C05460=1033.712,281.637,380.636,171.073,44.335,158.518
C05461=1033.719,281.885,380.604,171.077,44.336,158.519
C05462=1033.726,282.133,380.573,171.081,44.336,158.519
C05463=1033.732,282.381,380.541,171.084,44.336,158.520
C05464=1033.739,282.629,380.510,171.088,44.337,158.520
C05465=1033.746,282.877,380.479,171.092,44.337,158.521
C05466=1033.753,283.125,380.447,171.095,44.338,158.521
C05467=1033.759,283.373,380.416,171.100,44.338,158.522
C05468=1033.766,283.621,380.384,171.103,44.339,158.522
C05469=1033.773,283.869,380.353,171.107,44.340,158.522
C05470=1033.779,284.116,380.321,171.111,44.339,158.523
C05471=1033.786,284.364,380.290,171.115,44.340,158.523
C05472=1033.793,284.612,380.259,171.118,44.341,158.524
C05473=1033.800,284.860,380.226,171.123,44.341,158.524
C05474=1033.807,285.107,380.195,171.126,44.342,158.525
C05475=1033.814,285.356,380.163,171.130,44.342,158.525
C05476=1033.821,285.604,380.132,171.134,44.343,158.526
C05477=1033.827,285.852,380.100,171.138,44.343,158.526
C05478=1033.834,286.100,380.069,171.141,44.344,158.527
C05479=1033.841,286.347,380.037,171.146,44.344,158.527
C05480=1033.848,286.595,380.005,171.149,44.344,158.527
C05481=1033.855,286.843,379.974,171.154,44.345,158.528
C05482=1033.861,287.091,379.942,171.157,44.346,158.529
C05483=1033.869,287.339,379.910,171.161,44.346,158.529
C05484=1033.876,287.587,379.879,171.165,44.347,158.530
C05485=1033.882,287.835,379.846,171.169,44.348,158.530
C05486=1033.889,288.082,379.814,171.172,44.348,158.530
C05487=1033.895,288.330,379.783,171.177,44.349,158.531
C05488=1033.902,288.578,379.751,171.181,44.349,158.531
C05489=1033.910,288.826,379.719,171.185,44.350,158.532
C05490=1033.917,289.074,379.688,171.189,44.350,158.532
C05491=1033.923,289.321,379.655,171.192,44.351,158.533
C05492=1033.930,289.569,379.623,171.197,44.351,158.533
C05493=1033.937,289.817,379.591,171.200,44.352,158.534
C05494=1033.944,290.065,379.559,171.204,44.352,158.534
C05495=1033.950,290.313,379.527,171.208,44.353,158.535
C05496=1033.957,290.561,379.495,171.212,44.354,158.535
C05497=1033.964,290.808,379.463,171.216,44.354,158.536
C05498=1033.971,291.056,379.432,171.220,44.355,158.536
C05499=1033.981,291.421,379.384,171.226,44.356,158.537
C05500=1033.991,291.785,379.336,171.232,44.357,158.538
C05501=1034.001,292.150,379.289,171.238,44.358,158.539
C05502=1034.012,292.514,379.242,171.243,44.359,158.539
C05503=1034.018,292.762,379.209,171.248,44.359,158.540
C05504=1034.025,293.010,379.178,171.251,44.360,158.540
C05505=1034.032,293.258,379.145,171.256,44.361,158.541
C05506=1034.039,293.505,379.113,171.260,44.362,158.542
C05507=1034.045,293.753,379.081,171.263,44.362,158.542
C05508=1034.052,294.002,379.048,171.268,44.363,158.542
C05509=1034.059,294.249,379.016,171.271,44.364,158.543
C05510=1034.066,294.496,378.984,171.276,44.364,158.544
C05511=1034.072,294.744,378.952,171.279,44.365,158.544
C05512=1034.080,294.992,378.919,171.284,44.366,158.545
C05513=1034.086,295.240,378.887,171.288,44.366,158.545
C05514=1034.092,295.488,378.854,171.293,44.368,158.546
C05515=1034.099,295.736,378.821,171.296,44.368,158.546
C05516=1034.106,295.983,378.789,171.300,44.369,158.547
C05517=1034.113,296.231,378.756,171.304,44.370,158.547
C05518=1034.120,296.479,378.723,171.308,44.370,158.548
C05519=1034.127,296.726,378.691,171.313,44.371,158.549
C05520=1034.133,296.974,378.658,171.316,44.372,158.549
C05521=1034.140,297.222,378.625,171.321,44.373,158.550
C05522=1034.146,297.470,378.592,171.324,44.374,158.550
C05523=1034.153,297.717,378.560,171.329,44.375,158.551
C05524=1034.160,297.965,378.527,171.333,44.375,158.551
C05525=1034.167,298.212,378.493,171.338,44.376,158.552
C05526=1034.174,298.460,378.461,171.341,44.377,158.553
C05527=1034.180,298.708,378.428,171.345,44.378,158.553
C05528=1034.187,298.955,378.395,171.350,44.379,158.554
C05529=1034.194,299.204,378.362,171.353,44.380,158.554
C05530=1034.201,299.451,378.330,171.358,44.381,158.555
C05531=1034.208,299.699,378.297,171.361,44.381,158.555
C05532=1034.214,299.946,378.263,171.366,44.382,158.556
C05533=1034.220,300.194,378.231,171.371,44.383,158.557
C05534=1034.228,300.442,378.198,171.374,44.384,158.557
C05535=1034.234,300.690,378.165,171.379,44.385,158.558
C05536=1034.242,300.937,378.132,171.383,44.386,158.558
C05537=1034.248,301.185,378.099,171.387,44.387,158.559
C05538=1034.256,301.433,378.066,171.391,44.388,158.560
C05539=1034.262,301.680,378.033,171.396,44.388,158.560
C05540=1034.269,301.928,378.000,171.400,44.389,158.561
C05541=1034.275,302.176,377.967,171.404,44.390,158.561
C05542=1034.283,302.424,377.935,171.408,44.391,158.562
C05543=1034.290,302.671,377.901,171.413,44.392,158.563
C05544=1034.296,302.919,377.868,171.416,44.393,158.563
C05545=1034.303,303.166,377.835,171.421,44.394,158.564
C05546=1034.311,303.414,377.802,171.426,44.395,158.564
C05547=1034.318,303.662,377.769,171.429,44.396,158.565
C05548=1034.324,303.909,377.735,171.434,44.396,158.565
C05549=1034.331,304.157,377.702,171.438,44.397,158.566
C05550=1034.338,304.404,377.669,171.442,44.398,158.567
C05551=1034.345,304.652,377.636,171.447,44.399,158.567
C05552=1034.352,304.900,377.603,171.451,44.400,158.568
C05553=1034.359,305.148,377.570,171.456,44.401,158.569
C05554=1034.366,305.395,377.536,171.459,44.402,158.569
C05555=1034.378,305.776,377.485,171.466,44.404,158.570
C05556=1034.388,306.158,377.434,171.473,44.405,158.571
C05557=1034.399,306.539,377.383,171.480,44.407,158.572
C05558=1034.410,306.921,377.331,171.487,44.408,158.573
C05559=1034.417,307.169,377.298,171.490,44.409,158.574
C05560=1034.423,307.416,377.265,171.495,44.410,158.574
C05561=1034.431,307.663,377.231,171.500,44.411,158.575
C05562=1034.438,307.911,377.198,171.503,44.412,158.575
C05563=1034.445,308.159,377.164,171.508,44.413,158.576
C05564=1034.452,308.406,377.131,171.513,44.414,158.577
C05565=1034.459,308.654,377.098,171.517,44.415,158.577
C05566=1034.467,308.902,377.065,171.522,44.416,158.578
C05567=1034.474,309.149,377.031,171.526,44.417,158.579
C05568=1034.481,309.396,376.997,171.531,44.418,158.579
C05569=1034.488,309.645,376.964,171.535,44.419,158.580
C05570=1034.495,309.892,376.930,171.539,44.420,158.581
C05571=1034.503,310.140,376.897,171.544,44.421,158.581
C05572=1034.510,310.387,376.863,171.548,44.422,158.582
C05573=1034.517,310.635,376.829,171.553,44.423,158.583
C05574=1034.524,310.882,376.796,171.557,44.424,158.583
C05575=1034.531,311.130,376.762,171.562,44.425,158.584
C05576=1034.538,311.378,376.730,171.566,44.426,158.585
C05577=1034.546,311.625,376.696,171.571,44.427,158.585
C05578=1034.552,311.873,376.661,171.576,44.428,158.586
C05579=1034.559,312.120,376.627,171.580,44.430,158.587
C05580=1034.566,312.368,376.593,171.584,44.431,158.587
C05581=1034.573,312.615,376.559,171.589,44.432,158.588
C05582=1034.580,312.863,376.525,171.593,44.433,158.589
C05583=1034.586,313.111,376.491,171.598,44.435,158.589
C05584=1034.593,313.357,376.457,171.603,44.436,158.590
C05585=1034.600,313.605,376.422,171.606,44.437,158.591
C05586=1034.607,313.853,376.388,171.611,44.438,158.591
C05587=1034.614,314.101,376.355,171.616,44.439,158.592
C05588=1034.621,314.348,376.319,171.621,44.440,158.593
C05589=1034.628,314.596,376.286,171.625,44.442,158.594
C05590=1034.635,314.844,376.251,171.630,44.443,158.594
C05591=1034.641,315.090,376.217,171.635,44.444,158.595
C05592=1034.649,315.338,376.183,171.638,44.445,158.596
C05593=1034.655,315.586,376.149,171.643,44.447,158.597
C05594=1034.663,315.833,376.114,171.648,44.448,158.597
C05595=1034.669,316.081,376.080,171.653,44.449,158.598
C05596=1034.677,316.328,376.045,171.657,44.451,158.599
C05597=1034.684,316.576,376.011,171.662,44.452,158.599
C05598=1034.690,316.823,375.977,171.667,44.453,158.600
C05599=1034.698,317.071,375.942,171.671,44.454,158.601
C05600=1034.704,317.319,375.908,171.675,44.456,158.602
C05601=1034.712,317.566,375.874,171.680,44.457,158.602
C05602=1034.718,317.814,375.839,171.685,44.458,158.603
C05603=1034.726,318.061,375.805,171.690,44.460,158.604
C05604=1034.733,318.308,375.771,171.695,44.461,158.605
C05605=1034.740,318.556,375.736,171.699,44.463,158.605
C05606=1034.747,318.803,375.702,171.704,44.463,158.606
C05607=1034.754,319.051,375.667,171.709,44.465,158.607
C05608=1034.761,319.298,375.632,171.713,44.466,158.608
C05609=1034.768,319.546,375.598,171.718,44.468,158.608
C05610=1034.775,319.793,375.563,171.723,44.469,158.609
C05611=1034.787,320.179,375.509,171.730,44.471,158.610
C05612=1034.797,320.566,375.455,171.737,44.473,158.611
C05613=1034.809,320.952,375.401,171.745,44.475,158.613
C05614=1034.820,321.338,375.346,171.753,44.477,158.614
C05615=1034.827,321.585,375.312,171.757,44.479,158.615
C05616=1034.834,321.834,375.277,171.762,44.480,158.615
C05617=1034.842,322.081,375.243,171.767,44.481,158.616
C05618=1034.848,322.328,375.207,171.772,44.483,158.617
C05619=1034.856,322.575,375.173,171.777,44.485,158.618
C05620=1034.863,322.822,375.138,171.782,44.485,158.618
C05621=1034.871,323.070,375.103,171.787,44.487,158.619
C05622=1034.878,323.318,375.069,171.792,44.489,158.620
C05623=1034.885,323.566,375.034,171.795,44.490,158.621
C05624=1034.892,323.813,374.999,171.800,44.491,158.622
C05625=1034.900,324.061,374.964,171.805,44.493,158.622
C05626=1034.907,324.308,374.929,171.810,44.494,158.623
C05627=1034.914,324.555,374.894,171.815,44.496,158.624
C05628=1034.922,324.803,374.859,171.820,44.497,158.625
C05629=1034.929,325.050,374.824,171.825,44.499,158.626
C05630=1034.936,325.297,374.790,171.830,44.500,158.626
C05631=1034.944,325.545,374.754,171.835,44.501,158.627
C05632=1034.951,325.792,374.720,171.840,44.503,158.628
C05633=1034.958,326.040,374.684,171.845,44.504,158.629
C05634=1034.966,326.287,374.650,171.850,44.506,158.630
C05635=1034.973,326.535,374.614,171.855,44.507,158.630
C05636=1034.981,326.783,374.579,171.860,44.509,158.631
C05637=1034.988,327.030,374.544,171.865,44.510,158.632
C05638=1034.996,327.276,374.509,171.870,44.512,158.633
C05639=1035.003,327.524,374.474,171.875,44.513,158.634
C05640=1035.010,327.772,374.439,171.880,44.515,158.635
C05641=1035.018,328.020,374.404,171.885,44.516,158.635
C05642=1035.025,328.267,374.369,171.890,44.517,158.636
C05643=1035.033,328.514,374.333,171.895,44.519,158.637
C05644=1035.040,328.761,374.298,171.900,44.521,158.638
C05645=1035.047,329.008,374.262,171.905,44.523,158.639
C05646=1035.054,329.256,374.226,171.910,44.524,158.640
C05647=1035.061,329.504,374.191,171.915,44.526,158.640
C05648=1035.069,329.751,374.155,171.920,44.528,158.641
C05649=1035.075,329.998,374.120,171.925,44.529,158.642
C05650=1035.083,330.246,374.084,171.930,44.531,158.643
C05651=1035.090,330.493,374.048,171.935,44.532,158.644
C05652=1035.097,330.741,374.012,171.941,44.534,158.645
C05653=1035.105,330.988,373.978,171.946,44.536,158.646
C05654=1035.113,331.235,373.941,171.951,44.538,158.646
C05655=1035.120,331.482,373.906,171.956,44.539,158.647
C05656=1035.127,331.730,373.870,171.961,44.541,158.648
C05657=1035.134,331.977,373.834,171.966,44.543,158.649
C05658=1035.142,332.225,373.799,171.971,44.544,158.650
C05659=1035.149,332.472,373.763,171.976,44.546,158.651
C05660=1035.156,332.719,373.727,171.981,44.548,158.652
C05661=1035.164,332.967,373.691,171.986,44.550,158.653
C05662=1035.171,333.214,373.655,171.991,44.551,158.654
C05663=1035.178,333.461,373.619,171.996,44.553,158.654
C05664=1035.185,333.708,373.583,172.002,44.555,158.655
C05665=1035.193,333.956,373.548,172.007,44.557,158.656
C05666=1035.201,334.204,373.512,172.012,44.558,158.657
C05667=1035.212,334.585,373.456,172.021,44.561,158.659
C05668=1035.223,334.966,373.401,172.028,44.564,158.660
C05669=1035.235,335.348,373.345,172.036,44.567,158.661
C05670=1035.246,335.729,373.289,172.045,44.570,158.663
C05671=1035.254,335.977,373.252,172.050,44.571,158.664
C05672=1035.261,336.224,373.216,172.055,44.573,158.665
C05673=1035.268,336.471,373.180,172.061,44.575,158.666
C05674=1035.275,336.719,373.143,172.066,44.577,158.667
C05675=1035.283,336.966,373.107,172.071,44.579,158.668
C05676=1035.290,337.213,373.071,172.076,44.581,158.668
C05677=1035.298,337.460,373.035,172.082,44.583,158.670
C05678=1035.305,337.708,372.999,172.088,44.585,158.671
C05679=1035.312,337.956,372.962,172.093,44.586,158.671
C05680=1035.319,338.202,372.926,172.098,44.588,158.672
C05681=1035.327,338.449,372.889,172.103,44.591,158.673
C05682=1035.335,338.697,372.853,172.108,44.592,158.674
C05683=1035.343,338.944,372.817,172.114,44.594,158.675
C05684=1035.350,339.192,372.780,172.120,44.596,158.676
C05685=1035.357,339.438,372.744,172.125,44.598,158.677
C05686=1035.365,339.685,372.707,172.130,44.600,158.678
C05687=1035.372,339.933,372.671,172.135,44.602,158.679
C05688=1035.379,340.181,372.634,172.142,44.604,158.680
C05689=1035.387,340.427,372.597,172.147,44.606,158.681
C05690=1035.395,340.675,372.561,172.152,44.608,158.682
C05691=1035.403,340.922,372.524,172.157,44.610,158.683
C05692=1035.410,341.170,372.487,172.164,44.612,158.684
C05693=1035.417,341.416,372.452,172.169,44.614,158.685
C05694=1035.425,341.663,372.415,172.174,44.616,158.686
C05695=1035.432,341.910,372.377,172.179,44.618,158.687
C05696=1035.440,342.158,372.341,172.185,44.620,158.688
C05697=1035.447,342.405,372.303,172.191,44.622,158.689
C05698=1035.455,342.652,372.267,172.196,44.624,158.690
C05699=1035.462,342.899,372.230,172.201,44.626,158.691
C05700=1035.470,343.146,372.193,172.207,44.628,158.692
C05701=1035.477,343.394,372.156,172.213,44.631,158.693
C05702=1035.485,343.641,372.119,172.219,44.633,158.694
C05703=1035.492,343.888,372.081,172.224,44.635,158.696
C05704=1035.500,344.135,372.045,172.230,44.637,158.697
C05705=1035.507,344.382,372.008,172.235,44.639,158.698
C05706=1035.515,344.629,371.971,172.241,44.641,158.699
C05707=1035.522,344.876,371.933,172.246,44.643,158.700
C05708=1035.530,345.124,371.897,172.252,44.645,158.701
C05709=1035.537,345.371,371.859,172.258,44.647,158.702
C05710=1035.545,345.618,371.823,172.263,44.650,158.703
C05711=1035.552,345.865,371.785,172.269,44.652,158.704
C05712=1035.560,346.112,371.748,172.275,44.654,158.705
C05713=1035.568,346.359,371.711,172.280,44.656,158.706
C05714=1035.575,346.606,371.673,172.287,44.659,158.707
C05715=1035.583,346.854,371.636,172.292,44.661,158.708
C05716=1035.591,347.101,371.598,172.297,44.663,158.709
C05717=1035.599,347.348,371.561,172.303,44.665,158.710
C05718=1035.606,347.595,371.524,172.309,44.668,158.712
C05719=1035.614,347.842,371.487,172.315,44.670,158.713
C05720=1035.621,348.089,371.449,172.321,44.672,158.714
C05721=1035.629,348.337,371.411,172.326,44.675,158.715
C05722=1035.637,348.583,371.374,172.332,44.676,158.716
C05723=1035.649,348.961,371.317,172.342,44.680,158.717
C05724=1035.660,349.339,371.259,172.350,44.684,158.719
C05725=1035.672,349.718,371.202,172.359,44.687,158.721
C05726=1035.684,350.096,371.144,172.368,44.691,158.723
C05727=1035.691,350.343,371.107,172.374,44.693,158.724
C05728=1035.699,350.590,371.068,172.380,44.696,158.725
C05729=1035.706,350.837,371.030,172.385,44.698,158.726
C05730=1035.715,351.084,370.993,172.391,44.700,158.727
C05731=1035.722,351.331,370.955,172.398,44.703,158.728
C05732=1035.730,351.579,370.917,172.403,44.705,158.729
C05733=1035.737,351.825,370.879,172.409,44.708,158.731
C05734=1035.745,352.072,370.842,172.415,44.710,158.732
C05735=1035.753,352.319,370.803,172.422,44.713,158.733
C05736=1035.761,352.566,370.766,172.427,44.715,158.734
C05737=1035.769,352.813,370.728,172.433,44.717,158.735
C05738=1035.776,353.060,370.689,172.439,44.720,158.737
C05739=1035.784,353.307,370.652,172.446,44.723,158.738
C05740=1035.792,353.554,370.613,172.451,44.725,158.739
C05741=1035.799,353.801,370.575,172.457,44.727,158.740
C05742=1035.807,354.049,370.537,172.463,44.730,158.741
C05743=1035.815,354.295,370.499,172.470,44.732,158.743
C05744=1035.823,354.541,370.461,172.475,44.735,158.744
C05745=1035.831,354.789,370.423,172.482,44.738,158.745
C05746=1035.838,355.036,370.385,172.488,44.740,158.746
C05747=1035.847,355.283,370.346,172.494,44.742,158.747
C05748=1035.854,355.529,370.308,172.500,44.745,158.748
C05749=1035.862,355.777,370.270,172.506,44.747,158.750
C05750=1035.869,356.024,370.232,172.512,44.750,158.751
C05751=1035.878,356.271,370.193,172.518,44.752,158.752
C05752=1035.885,356.518,370.155,172.524,44.755,158.753
C05753=1035.893,356.765,370.117,172.531,44.758,158.755
C05754=1035.901,357.012,370.078,172.537,44.761,158.756
C05755=1035.909,357.258,370.040,172.543,44.763,158.757
C05756=1035.917,357.506,370.001,172.549,44.766,158.758
C05757=1035.925,357.752,369.963,172.555,44.768,158.760
C05758=1035.933,357.999,369.923,172.562,44.771,158.761
C05759=1035.941,358.245,369.885,172.568,44.774,158.762
C05760=1035.949,358.493,369.847,172.574,44.777,158.763
C05761=1035.957,358.740,369.808,172.581,44.779,158.765
C05762=1035.965,358.986,369.770,172.587,44.782,158.766
C05763=1035.973,359.233,369.731,172.593,44.784,158.767
C05764=1035.981,359.480,369.692,172.600,44.787,158.769
C05765=1035.988,359.727,369.653,172.606,44.790,158.770
C05766=1035.996,359.974,369.614,172.612,44.792,158.771
C05767=1036.005,360.221,369.575,172.619,44.795,158.772
C05768=1036.012,360.467,369.537,172.625,44.798,158.774
C05769=1036.020,360.714,369.498,172.631,44.801,158.775
C05770=1036.029,360.961,369.459,172.638,44.804,158.776
C05771=1036.037,361.208,369.420,172.644,44.807,158.778
C05772=1036.044,361.455,369.382,172.650,44.809,158.779
C05773=1036.052,361.702,369.342,172.657,44.812,158.780
C05774=1036.061,361.948,369.303,172.664,44.815,158.782
C05775=1036.069,362.196,369.264,172.670,44.818,158.783
C05776=1036.076,362.442,369.225,172.676,44.821,158.784
C05777=1036.084,362.689,369.186,172.683,44.824,158.786
C05778=1036.092,362.936,369.146,172.690,44.827,158.787
C05779=1036.104,363.320,369.086,172.699,44.831,158.789
C05780=1036.117,363.704,369.024,172.709,44.836,158.791
C05781=1036.129,364.089,368.963,172.720,44.840,158.793
C05782=1036.142,364.473,368.901,172.730,44.845,158.795
C05783=1036.150,364.720,368.862,172.736,44.848,158.797
C05784=1036.158,364.967,368.822,172.743,44.851,158.798
C05785=1036.166,365.214,368.783,172.750,44.854,158.800
C05786=1036.174,365.461,368.743,172.757,44.857,158.801
C05787=1036.182,365.707,368.704,172.763,44.860,158.802
C05788=1036.191,365.954,368.665,172.770,44.863,158.804
C05789=1036.199,366.201,368.625,172.777,44.866,158.805
C05790=1036.207,366.447,368.586,172.783,44.869,158.807
C05791=1036.215,366.694,368.546,172.790,44.872,158.808
C05792=1036.223,366.941,368.506,172.797,44.875,158.809
C05793=1036.231,367.188,368.466,172.804,44.878,158.811
C05794=1036.240,367.434,368.426,172.811,44.881,158.812
C05795=1036.248,367.680,368.387,172.817,44.884,158.814
C05796=1036.256,367.927,368.347,172.823,44.887,158.815
C05797=1036.264,368.174,368.308,172.830,44.890,158.817
C05798=1036.272,368.421,368.268,172.837,44.893,158.818
C05799=1036.281,368.667,368.228,172.844,44.897,158.819
C05800=1036.289,368.913,368.189,172.851,44.900,158.821
C05801=1036.297,369.160,368.149,172.858,44.903,158.822
C05802=1036.306,369.408,368.109,172.865,44.906,158.824
C05803=1036.314,369.654,368.068,172.872,44.909,158.825
C05804=1036.323,369.900,368.029,172.879,44.912,158.827
C05805=1036.331,370.147,367.988,172.886,44.916,158.828
C05806=1036.338,370.394,367.948,172.892,44.919,158.830
C05807=1036.347,370.640,367.908,172.900,44.922,158.831
C05808=1036.355,370.887,367.868,172.906,44.925,158.833
C05809=1036.363,371.134,367.827,172.914,44.929,158.834
C05810=1036.371,371.380,367.788,172.920,44.932,158.836
C05811=1036.380,371.626,367.747,172.928,44.936,158.837
C05812=1036.388,371.873,367.707,172.934,44.939,158.839
C05813=1036.396,372.120,367.667,172.942,44.942,158.840
C05814=1036.404,372.367,367.626,172.948,44.945,158.842
C05815=1036.413,372.613,367.586,172.956,44.949,158.843
C05816=1036.421,372.859,367.545,172.962,44.952,158.845
C05817=1036.430,373.106,367.504,172.970,44.955,158.846
C05818=1036.437,373.353,367.464,172.977,44.959,158.848
C05819=1036.446,373.599,367.424,172.984,44.962,158.850
C05820=1036.455,373.846,367.383,172.992,44.965,158.851
C05821=1036.463,374.092,367.343,172.999,44.969,158.853
C05822=1036.471,374.338,367.302,173.006,44.972,158.854
C05823=1036.479,374.585,367.261,173.013,44.976,158.856
C05824=1036.488,374.831,367.221,173.020,44.979,158.857
C05825=1036.497,375.078,367.180,173.027,44.983,158.859
C05826=1036.505,375.324,367.139,173.034,44.986,158.861
C05827=1036.514,375.571,367.098,173.041,44.990,158.862
C05828=1036.522,375.817,367.058,173.049,44.993,158.864
C05829=1036.530,376.064,367.018,173.057,44.997,158.865
C05830=1036.539,376.311,366.977,173.064,45.000,158.867
C05831=1036.547,376.556,366.935,173.071,45.004,158.869
C05832=1036.556,376.803,366.894,173.078,45.007,158.870
C05833=1036.565,377.050,366.854,173.086,45.011,158.872
C05834=1036.573,377.296,366.813,173.093,45.014,158.874
C05835=1036.587,377.701,366.745,173.106,45.020,158.876
C05836=1036.602,378.106,366.678,173.117,45.026,158.879
C05837=1036.615,378.511,366.610,173.130,45.032,158.882
C05838=1036.629,378.915,366.542,173.142,45.038,158.884
C05839=1036.638,379.162,366.501,173.150,45.041,158.886
C05840=1036.647,379.409,366.460,173.157,45.046,158.888
C05841=1036.655,379.654,366.418,173.164,45.049,158.890
C05842=1036.664,379.901,366.377,173.172,45.052,158.891
C05843=1036.673,380.148,366.336,173.180,45.056,158.893
C05844=1036.681,380.393,366.294,173.187,45.060,158.895
C05845=1036.690,380.640,366.253,173.195,45.064,158.896
C05846=1036.698,380.887,366.211,173.203,45.067,158.898
C05847=1036.706,381.133,366.170,173.210,45.072,158.900
C05848=1036.715,381.379,366.128,173.218,45.075,158.902
C05849=1036.724,381.625,366.086,173.226,45.079,158.903
C05850=1036.733,381.872,366.045,173.233,45.083,158.905
C05851=1036.741,382.117,366.003,173.241,45.087,158.907
C05852=1036.750,382.364,365.961,173.249,45.091,158.909
C05853=1036.758,382.611,365.920,173.257,45.094,158.910
C05854=1036.767,382.857,365.878,173.264,45.099,158.912
C05855=1036.776,383.103,365.836,173.272,45.103,158.914
C05856=1036.785,383.349,365.794,173.280,45.106,158.916
C05857=1036.793,383.595,365.753,173.287,45.110,158.917
C05858=1036.802,383.842,365.711,173.296,45.114,158.919
C05859=1036.811,384.088,365.669,173.303,45.118,158.921
C05860=1036.819,384.335,365.627,173.312,45.122,158.923
C05861=1036.828,384.581,365.585,173.319,45.126,158.925
C05862=1036.838,384.827,365.543,173.328,45.130,158.927
C05863=1036.847,385.073,365.501,173.335,45.134,158.928
C05864=1036.856,385.319,365.459,173.343,45.138,158.930
C05865=1036.865,385.565,365.417,173.351,45.142,158.932
C05866=1036.873,385.812,365.375,173.359,45.146,158.934
C05867=1036.882,386.058,365.333,173.368,45.150,158.936
C05868=1036.891,386.304,365.290,173.375,45.154,158.937
C05869=1036.900,386.550,365.249,173.384,45.157,158.939
C05870=1036.910,386.797,365.206,173.391,45.162,158.941
C05871=1036.919,387.043,365.164,173.400,45.166,158.943
C05872=1036.927,387.289,365.121,173.408,45.170,158.945
C05873=1036.936,387.536,365.079,173.416,45.174,158.947
C05874=1036.946,387.781,365.037,173.424,45.178,158.949
C05875=1036.954,388.028,364.995,173.432,45.182,158.951
C05876=1036.963,388.274,364.952,173.440,45.187,158.953
C05877=1036.973,388.520,364.910,173.449,45.191,158.954
C05878=1036.981,388.766,364.866,173.457,45.195,158.956
C05879=1036.991,389.012,364.824,173.465,45.199,158.958
C05880=1036.999,389.258,364.781,173.474,45.204,158.960
C05881=1037.008,389.504,364.739,173.481,45.208,158.962
C05882=1037.017,389.751,364.696,173.490,45.212,158.964
C05883=1037.026,389.997,364.653,173.499,45.216,158.966
C05884=1037.036,390.243,364.611,173.507,45.220,158.968
C05885=1037.045,390.489,364.568,173.515,45.225,158.970
C05886=1037.054,390.735,364.525,173.524,45.229,158.972
C05887=1037.062,390.981,364.482,173.532,45.234,158.974
C05888=1037.072,391.226,364.439,173.541,45.238,158.976
C05889=1037.081,391.473,364.396,173.548,45.242,158.978
C05890=1037.090,391.719,364.353,173.557,45.246,158.980
C05891=1037.098,391.939,364.315,173.565,45.250,158.982
C05892=1037.107,392.158,364.275,173.573,45.254,158.984
C05893=1037.115,392.378,364.237,173.581,45.258,158.985
C05894=1037.123,392.598,364.198,173.588,45.262,158.987
C05895=1037.131,392.818,364.160,173.595,45.266,158.989
C05896=1037.139,393.036,364.121,173.603,45.270,158.991
C05897=1037.148,393.257,364.083,173.611,45.274,158.993
C05898=1037.155,393.476,364.044,173.619,45.278,158.995
C05899=1037.165,393.722,364.001,173.628,45.283,158.997
C05900=1037.174,393.968,363.958,173.637,45.288,158.999
C05901=1037.183,394.214,363.914,173.645,45.292,159.001
C05902=1037.193,394.461,363.871,173.654,45.296,159.003
C05903=1037.202,394.706,363.827,173.662,45.301,159.005
C05904=1037.212,394.952,363.784,173.671,45.306,159.007
C05905=1037.220,395.198,363.741,173.680,45.310,159.009
C05906=1037.230,395.444,363.696,173.689,45.315,159.011
C05907=1037.238,395.690,363.653,173.697,45.319,159.013
C05908=1037.248,395.936,363.609,173.706,45.324,159.016
C05909=1037.258,396.182,363.565,173.715,45.329,159.018
C05910=1037.267,396.427,363.521,173.724,45.334,159.020
C05911=1037.276,396.673,363.477,173.733,45.339,159.022
C05912=1037.285,396.920,363.434,173.742,45.343,159.024
C05913=1037.294,397.165,363.390,173.751,45.348,159.026
C05914=1037.304,397.411,363.347,173.760,45.353,159.029
C05915=1037.314,397.657,363.302,173.770,45.357,159.031
C05916=1037.323,397.903,363.258,173.779,45.362,159.033
C05917=1037.333,398.149,363.214,173.788,45.367,159.035
C05918=1037.342,398.394,363.170,173.797,45.372,159.037
C05919=1037.352,398.640,363.126,173.806,45.376,159.040
C05920=1037.361,398.886,363.082,173.815,45.381,159.042
C05921=1037.371,399.132,363.037,173.824,45.386,159.044
C05922=1037.380,399.378,362.993,173.834,45.391,159.046
C05923=1037.390,399.624,362.949,173.843,45.396,159.049
C05924=1037.399,399.870,362.904,173.852,45.401,159.051
C05925=1037.409,400.116,362.860,173.861,45.406,159.053
C05926=1037.419,400.361,362.815,173.870,45.410,159.055
C05927=1037.428,400.608,362.771,173.880,45.416,159.058
C05928=1037.438,400.853,362.726,173.889,45.420,159.060
C05929=1037.447,401.099,362.682,173.898,45.425,159.062
C05930=1037.457,401.345,362.637,173.908,45.431,159.065
C05931=1037.467,401.590,362.593,173.918,45.435,159.067
C05932=1037.476,401.836,362.549,173.927,45.440,159.069
C05933=1037.486,402.082,362.504,173.936,45.446,159.072
C05934=1037.495,402.327,362.459,173.945,45.451,159.074
C05935=1037.505,402.573,362.414,173.956,45.456,159.076
C05936=1037.515,402.819,362.370,173.965,45.461,159.079
C05937=1037.524,403.064,362.325,173.974,45.466,159.081
C05938=1037.535,403.311,362.280,173.984,45.471,159.084
C05939=1037.544,403.557,362.235,173.994,45.477,159.086
C05940=1037.553,403.802,362.190,174.004,45.481,159.088
C05941=1037.563,404.048,362.145,174.013,45.487,159.091
C05942=1037.573,404.292,362.099,174.022,45.492,159.093
C05943=1037.583,404.539,362.054,174.033,45.497,159.096
C05944=1037.592,404.784,362.009,174.042,45.503,159.098
C05945=1037.602,405.030,361.964,174.052,45.508,159.100
C05946=1037.612,405.276,361.919,174.062,45.513,159.103
C05947=1037.622,405.521,361.873,174.072,45.518,159.105
C05948=1037.631,405.767,361.828,174.082,45.524,159.108
C05949=1037.642,406.013,361.783,174.092,45.529,159.110
C05950=1037.652,406.258,361.737,174.102,45.535,159.113
C05951=1037.663,406.565,361.680,174.114,45.541,159.116
C05952=1037.676,406.871,361.624,174.127,45.548,159.119
C05953=1037.688,407.176,361.567,174.139,45.554,159.122
C05954=1037.701,407.482,361.510,174.152,45.562,159.125
C05955=1037.711,407.728,361.464,174.162,45.567,159.128
C05956=1037.720,407.974,361.419,174.172,45.573,159.131
C05957=1037.731,408.219,361.373,174.182,45.578,159.133
C05958=1037.742,408.465,361.327,174.193,45.583,159.136
C05959=1037.751,408.710,361.281,174.202,45.589,159.138
C05960=1037.761,408.956,361.236,174.213,45.594,159.141
C05961=1037.772,409.202,361.190,174.223,45.600,159.143
C05962=1037.781,409.447,361.144,174.233,45.605,159.146
C05963=1037.792,409.693,361.098,174.243,45.611,159.149
C05964=1037.802,409.938,361.052,174.254,45.617,159.151
C05965=1037.812,410.184,361.006,174.265,45.622,159.154
C05966=1037.822,410.429,360.960,174.275,45.628,159.157
C05967=1037.833,410.675,360.914,174.285,45.634,159.159
C05968=1037.844,410.920,360.868,174.296,45.640,159.162
C05969=1037.853,411.166,360.822,174.306,45.645,159.165
C05970=1037.864,411.411,360.775,174.317,45.651,159.167
C05971=1037.874,411.656,360.729,174.328,45.657,159.170
C05972=1037.884,411.902,360.683,174.338,45.662,159.173
C05973=1037.895,412.147,360.636,174.349,45.668,159.175
C05974=1037.904,412.393,360.589,174.360,45.674,159.178
C05975=1037.915,412.638,360.543,174.371,45.680,159.181
C05976=1037.925,412.884,360.496,174.382,45.686,159.184
C05977=1037.936,413.129,360.450,174.392,45.691,159.186
C05978=1037.946,413.375,360.403,174.403,45.698,159.189
C05979=1037.956,413.620,360.356,174.414,45.703,159.192
C05980=1037.967,413.865,360.309,174.425,45.709,159.195
C05981=1037.977,414.111,360.263,174.436,45.715,159.198
C05982=1037.987,414.356,360.216,174.447,45.721,159.200
C05983=1038.005,414.755,360.139,174.464,45.731,159.205
C05984=1038.022,415.154,360.063,174.482,45.741,159.210
C05985=1038.038,415.553,359.987,174.500,45.751,159.214
C05986=1038.056,415.951,359.910,174.518,45.761,159.219
C05987=1038.066,416.196,359.863,174.529,45.767,159.222
C05988=1038.077,416.441,359.817,174.541,45.773,159.225
C05989=1038.088,416.687,359.769,174.552,45.779,159.228
C05990=1038.099,416.932,359.721,174.564,45.785,159.231
C05991=1038.109,417.177,359.674,174.575,45.791,159.234
C05992=1038.120,417.423,359.627,174.587,45.797,159.237
C05993=1038.130,417.668,359.580,174.598,45.804,159.240
C05994=1038.142,417.913,359.531,174.609,45.810,159.243
C05995=1038.152,418.159,359.484,174.621,45.817,159.246
C05996=1038.163,418.404,359.436,174.632,45.823,159.249
C05997=1038.173,418.649,359.389,174.644,45.829,159.252
C05998=1038.184,418.894,359.341,174.656,45.835,159.255
C05999=1038.195,419.139,359.293,174.667,45.842,159.258
C06000=1038.206,419.384,359.246,174.679,45.848,159.261
C06001=1038.217,419.630,359.198,174.691,45.855,159.264
C06002=1038.227,419.874,359.150,174.703,45.861,159.267
C06003=1038.238,420.120,359.101,174.714,45.867,159.270
C06004=1038.249,420.365,359.053,174.726,45.874,159.273
C06005=1038.260,420.610,359.006,174.737,45.880,159.276
C06006=1038.271,420.856,358.957,174.750,45.887,159.279
C06007=1038.282,421.089,358.911,174.761,45.893,159.282
C06008=1038.291,421.323,358.865,174.772,45.899,159.285
C06009=1038.302,421.557,358.820,174.785,45.906,159.288
C06010=1038.313,421.791,358.773,174.796,45.912,159.291
C06011=1038.324,422.026,358.727,174.807,45.918,159.294
C06012=1038.334,422.259,358.681,174.819,45.925,159.298
C06013=1038.345,422.493,358.635,174.831,45.931,159.301
C06014=1038.355,422.727,358.588,174.842,45.937,159.304
C06015=1038.366,422.972,358.540,174.854,45.944,159.307
C06016=1038.377,423.218,358.492,174.867,45.951,159.310
C06017=1038.389,423.462,358.443,174.879,45.957,159.313
C06018=1038.400,423.708,358.394,174.892,45.964,159.317
C06019=1038.411,423.953,358.345,174.904,45.971,159.320
C06020=1038.422,424.198,358.297,174.916,45.978,159.323
C06021=1038.433,424.442,358.248,174.929,45.984,159.326
C06022=1038.445,424.687,358.199,174.941,45.991,159.330
C06023=1038.456,424.931,358.150,174.954,45.998,159.333
C06024=1038.467,425.178,358.101,174.967,46.006,159.337
C06025=1038.478,425.423,358.052,174.980,46.012,159.340
C06026=1038.490,425.667,358.003,174.992,46.019,159.343
C06027=1038.501,425.912,357.954,175.005,46.026,159.347
C06028=1038.513,426.157,357.905,175.018,46.033,159.350
C06029=1038.523,426.402,357.855,175.030,46.040,159.354
C06030=1038.535,426.647,357.806,175.043,46.047,159.357
C06031=1038.547,426.891,357.756,175.056,46.054,159.361
C06032=1038.558,427.136,357.707,175.069,46.061,159.364
C06033=1038.570,427.381,357.658,175.082,46.068,159.367
C06034=1038.581,427.626,357.609,175.096,46.076,159.371
C06035=1038.593,427.871,357.559,175.108,46.082,159.374
C06036=1038.604,428.116,357.510,175.121,46.090,159.378
C06037=1038.615,428.360,357.459,175.134,46.097,159.381
C06038=1038.627,428.605,357.410,175.148,46.104,159.385
C06039=1038.639,428.850,357.360,175.161,46.111,159.389
C06040=1038.650,429.095,357.309,175.174,46.119,159.392
C06041=1038.662,429.339,357.260,175.188,46.126,159.396
C06042=1038.673,429.584,357.210,175.202,46.134,159.400
C06043=1038.685,429.829,357.160,175.215,46.141,159.403
C06044=1038.697,430.074,357.109,175.229,46.148,159.407
C06045=1038.708,430.318,357.060,175.242,46.156,159.410
C06046=1038.721,430.563,357.009,175.256,46.163,159.414
C06047=1038.732,430.807,356.959,175.269,46.171,159.418
C06048=1038.744,431.052,356.909,175.283,46.178,159.421
C06049=1038.755,431.296,356.859,175.297,46.185,159.425
C06050=1038.767,431.541,356.809,175.311,46.193,159.429
C06051=1038.779,431.786,356.758,175.324,46.200,159.433
C06052=1038.792,432.031,356.707,175.338,46.208,159.436
C06053=1038.803,432.275,356.657,175.353,46.215,159.440
C06054=1038.815,432.520,356.607,175.366,46.223,159.444
C06055=1038.827,432.764,356.556,175.380,46.230,159.448
C06056=1038.839,433.009,356.505,175.395,46.238,159.452
C06057=1038.852,433.253,356.454,175.409,46.246,159.456
C06058=1038.863,433.498,356.404,175.423,46.254,159.459
C06059=1038.876,433.743,356.353,175.437,46.261,159.463
C06060=1038.887,433.986,356.302,175.452,46.269,159.467
C06061=1038.899,434.231,356.252,175.466,46.277,159.471
C06062=1038.912,434.476,356.201,175.481,46.284,159.475
C06063=1038.925,434.721,356.149,175.495,46.292,159.479
C06064=1038.937,434.965,356.098,175.510,46.300,159.483
C06065=1038.949,435.209,356.047,175.524,46.308,159.487
C06066=1038.961,435.454,355.996,175.539,46.316,159.491
C06067=1038.973,435.692,355.946,175.553,46.324,159.495
C06068=1038.986,435.931,355.895,175.567,46.331,159.499
C06069=1038.997,436.171,355.845,175.582,46.339,159.503
C06070=1039.009,436.409,355.795,175.596,46.347,159.507
C06071=1039.021,436.648,355.744,175.611,46.355,159.510
C06072=1039.033,436.886,355.694,175.625,46.362,159.515
C06073=1039.046,437.125,355.644,175.640,46.370,159.519
C06074=1039.058,437.364,355.593,175.655,46.378,159.523
C06075=1039.070,437.608,355.541,175.670,46.387,159.527
C06076=1039.083,437.852,355.490,175.686,46.394,159.531
C06077=1039.095,438.097,355.438,175.701,46.403,159.535
C06078=1039.107,438.341,355.386,175.715,46.411,159.539
C06079=1039.120,438.585,355.333,175.731,46.419,159.543
C06080=1039.133,438.829,355.282,175.746,46.427,159.548
C06081=1039.146,439.073,355.229,175.761,46.436,159.552
C06082=1039.158,439.317,355.177,175.777,46.444,159.556
C06083=1039.171,439.562,355.125,175.793,46.452,159.561
C06084=1039.184,439.805,355.073,175.809,46.460,159.565
C06085=1039.197,440.050,355.020,175.825,46.469,159.569
C06086=1039.209,440.294,354.968,175.840,46.477,159.574
C06087=1039.222,440.538,354.915,175.856,46.486,159.578
C06088=1039.235,440.783,354.863,175.871,46.494,159.582
C06089=1039.248,441.026,354.809,175.887,46.503,159.587
C06090=1039.260,441.270,354.757,175.904,46.511,159.591
C06091=1039.274,441.514,354.705,175.920,46.520,159.596
C06092=1039.287,441.759,354.652,175.936,46.529,159.600
C06093=1039.300,442.003,354.599,175.952,46.537,159.605
C06094=1039.313,442.247,354.546,175.968,46.546,159.609
C06095=1039.325,442.490,354.493,175.985,46.554,159.614
C06096=1039.338,442.734,354.441,176.001,46.563,159.618
C06097=1039.351,442.978,354.387,176.018,46.572,159.623
C06098=1039.364,443.222,354.334,176.034,46.580,159.627
C06099=1039.377,443.466,354.281,176.051,46.589,159.632
C06100=1039.391,443.710,354.228,176.067,46.598,159.636
C06101=1039.405,443.954,354.174,176.084,46.607,159.641
C06102=1039.418,444.198,354.121,176.100,46.615,159.646
C06103=1039.431,444.441,354.067,176.117,46.624,159.650
C06104=1039.444,444.684,354.015,176.135,46.633,159.655
C06105=1039.458,444.927,353.962,176.151,46.641,159.660
C06106=1039.473,445.171,353.910,176.168,46.651,159.664
C06107=1039.489,445.414,353.858,176.185,46.659,159.669
C06108=1039.505,445.658,353.807,176.203,46.667,159.673
C06109=1039.521,445.901,353.756,176.219,46.675,159.678
C06110=1039.538,446.145,353.706,176.237,46.683,159.683
C06111=1039.555,446.389,353.656,176.254,46.692,159.687
C06112=1039.574,446.633,353.606,176.271,46.700,159.692
C06113=1039.593,446.877,353.558,176.290,46.707,159.696
C06114=1039.612,447.121,353.509,176.307,46.715,159.701
C06115=1039.631,447.365,353.461,176.324,46.723,159.705
C06116=1039.652,447.610,353.414,176.343,46.730,159.710
C06117=1039.673,447.854,353.366,176.361,46.738,159.714
C06118=1039.695,448.099,353.320,176.379,46.745,159.719
C06119=1039.717,448.343,353.274,176.396,46.753,159.723
C06120=1039.740,448.588,353.228,176.414,46.760,159.727
C06121=1039.763,448.833,353.182,176.433,46.767,159.732
C06122=1039.787,449.078,353.137,176.452,46.774,159.736
C06123=1039.811,449.323,353.093,176.470,46.781,159.741
C06124=1039.836,449.568,353.050,176.489,46.788,159.745
C06125=1039.862,449.813,353.007,176.507,46.795,159.749
C06126=1039.888,450.058,352.963,176.526,46.801,159.754
C06127=1039.912,450.280,352.925,176.542,46.807,159.758
C06128=1039.937,450.502,352.887,176.559,46.813,159.762
C06129=1039.962,450.723,352.849,176.576,46.819,159.765
C06130=1039.987,450.945,352.811,176.594,46.824,159.769
C06131=1040.013,451.165,352.775,176.610,46.830,159.773
C06132=1040.040,451.387,352.738,176.627,46.836,159.777
C06133=1040.066,451.608,352.703,176.644,46.841,159.781
C06134=1040.094,451.829,352.667,176.663,46.846,159.785
C06135=1039.798,451.878,352.348,176.665,46.921,159.808
C06136=1039.771,451.664,352.382,176.648,46.916,159.804
C06137=1039.745,451.451,352.416,176.631,46.912,159.800
C06138=1039.719,451.237,352.452,176.615,46.906,159.797
C06139=1039.694,451.023,352.487,176.598,46.901,159.793
C06140=1039.669,450.808,352.523,176.582,46.895,159.789
C06141=1039.645,450.594,352.559,176.565,46.890,159.785
C06142=1039.621,450.380,352.596,176.549,46.884,159.782
C06143=1039.597,450.165,352.633,176.532,46.878,159.778
C06144=1039.570,449.920,352.676,176.514,46.872,159.774
C06145=1039.545,449.676,352.718,176.495,46.866,159.769
C06146=1039.520,449.430,352.762,176.477,46.859,159.765
C06147=1039.494,449.185,352.807,176.457,46.852,159.760
C06148=1039.470,448.940,352.851,176.440,46.845,159.756
C06149=1039.447,448.695,352.896,176.421,46.838,159.752
C06150=1039.424,448.451,352.941,176.402,46.831,159.747
C06151=1039.402,448.206,352.987,176.384,46.824,159.743
C06152=1039.380,447.961,353.034,176.367,46.816,159.739
C06153=1039.358,447.717,353.080,176.349,46.809,159.734
C06154=1039.338,447.472,353.128,176.330,46.802,159.729
C06155=1039.318,447.228,353.176,176.313,46.794,159.725
C06156=1039.297,446.984,353.225,176.295,46.786,159.720
C06157=1039.279,446.739,353.273,176.278,46.779,159.716
C06158=1039.260,446.495,353.323,176.260,46.771,159.711
C06159=1039.242,446.252,353.372,176.242,46.763,159.707
C06160=1039.225,446.008,353.422,176.224,46.755,159.702
C06161=1039.208,445.763,353.473,176.207,46.747,159.698
C06162=1039.192,445.520,353.523,176.190,46.738,159.693
C06163=1039.176,445.277,353.575,176.173,46.730,159.689
C06164=1039.162,445.033,353.627,176.155,46.722,159.684
C06165=1039.147,444.790,353.679,176.139,46.713,159.679
C06166=1039.133,444.546,353.732,176.122,46.704,159.675
C06167=1039.120,444.304,353.785,176.105,46.695,159.670
C06168=1039.106,444.061,353.839,176.088,46.687,159.665
C06169=1039.093,443.816,353.892,176.071,46.678,159.661
C06170=1039.079,443.572,353.945,176.055,46.670,159.656
C06171=1039.066,443.328,353.998,176.038,46.661,159.652
C06172=1039.053,443.084,354.051,176.021,46.652,159.647
C06173=1039.040,442.841,354.104,176.005,46.644,159.642
C06174=1039.027,442.597,354.158,175.989,46.635,159.638
C06175=1039.013,442.353,354.211,175.972,46.626,159.633
C06176=1039.000,442.109,354.264,175.956,46.618,159.629
C06177=1038.988,441.865,354.316,175.939,46.609,159.624
C06178=1038.975,441.621,354.369,175.923,46.601,159.620
C06179=1038.961,441.377,354.422,175.907,46.593,159.615
C06180=1038.948,441.133,354.474,175.891,46.584,159.611
C06181=1038.935,440.889,354.528,175.875,46.576,159.606
C06182=1038.923,440.645,354.580,175.859,46.567,159.602
C06183=1038.910,440.401,354.633,175.843,46.559,159.598
C06184=1038.897,440.156,354.686,175.828,46.551,159.593
C06185=1038.885,439.912,354.738,175.812,46.543,159.589
C06186=1038.872,439.668,354.790,175.795,46.534,159.585
C06187=1038.859,439.423,354.842,175.780,46.526,159.580
C06188=1038.847,439.179,354.894,175.764,46.517,159.576
C06189=1038.834,438.935,354.947,175.749,46.510,159.572
C06190=1038.821,438.691,354.998,175.733,46.501,159.568
C06191=1038.808,438.447,355.051,175.718,46.493,159.563
C06192=1038.796,438.203,355.103,175.702,46.485,159.559
C06193=1038.783,437.958,355.155,175.687,46.477,159.555
C06194=1038.770,437.714,355.206,175.672,46.469,159.551
C06195=1038.758,437.469,355.259,175.657,46.461,159.547
C06196=1038.746,437.230,355.309,175.642,46.453,159.543
C06197=1038.733,436.991,355.360,175.627,46.445,159.539
C06198=1038.721,436.752,355.411,175.612,46.437,159.534
C06199=1038.710,436.512,355.461,175.598,46.429,159.530
C06200=1038.697,436.274,355.511,175.583,46.422,159.527
C06201=1038.685,436.035,355.562,175.568,46.414,159.523
C06202=1038.674,435.795,355.612,175.554,46.407,159.519
C06203=1038.660,435.555,355.663,175.539,46.399,159.515
C06204=1038.649,435.311,355.714,175.525,46.391,159.511
C06205=1038.636,435.066,355.765,175.510,46.383,159.507
C06206=1038.624,434.822,355.816,175.495,46.375,159.503
C06207=1038.612,434.577,355.868,175.481,46.367,159.499
C06208=1038.600,434.333,355.918,175.466,46.360,159.495
C06209=1038.587,434.088,355.969,175.452,46.352,159.491
C06210=1038.575,433.844,356.020,175.437,46.344,159.487
C06211=1038.563,433.600,356.071,175.424,46.337,159.483
C06212=1038.551,433.355,356.122,175.410,46.329,159.479
C06213=1038.539,433.110,356.173,175.395,46.322,159.475
C06214=1038.527,432.865,356.223,175.381,46.314,159.472
C06215=1038.514,432.621,356.274,175.366,46.307,159.468
C06216=1038.503,432.377,356.324,175.353,46.299,159.464
C06217=1038.491,432.132,356.375,175.339,46.291,159.460
C06218=1038.478,431.888,356.425,175.324,46.284,159.456
C06219=1038.467,431.642,356.476,175.311,46.276,159.453
C06220=1038.455,431.399,356.526,175.297,46.269,159.449
C06221=1038.443,431.154,356.577,175.282,46.262,159.445
C06222=1038.431,430.909,356.627,175.269,46.254,159.442
C06223=1038.419,430.665,356.677,175.255,46.247,159.438
C06224=1038.408,430.420,356.728,175.242,46.240,159.434
C06225=1038.395,430.175,356.778,175.228,46.232,159.430
C06226=1038.384,429.931,356.828,175.215,46.225,159.427
C06227=1038.372,429.686,356.878,175.201,46.218,159.423
C06228=1038.360,429.442,356.928,175.188,46.211,159.420
C06229=1038.349,429.196,356.978,175.174,46.204,159.416
C06230=1038.337,428.952,357.028,175.160,46.196,159.412
C06231=1038.326,428.707,357.078,175.147,46.189,159.409
C06232=1038.314,428.462,357.127,175.133,46.182,159.405
C06233=1038.303,428.217,357.178,175.120,46.175,159.402
C06234=1038.292,427.973,357.227,175.107,46.167,159.398
C06235=1038.280,427.728,357.277,175.094,46.160,159.394
C06236=1038.268,427.483,357.326,175.081,46.153,159.391
C06237=1038.257,427.238,357.376,175.068,46.146,159.388
C06238=1038.245,426.993,357.425,175.055,46.139,159.384
C06239=1038.234,426.748,357.474,175.042,46.132,159.381
C06240=1038.222,426.504,357.523,175.029,46.125,159.377
C06241=1038.210,426.258,357.573,175.017,46.118,159.374
C06242=1038.199,426.014,357.622,175.003,46.111,159.370
C06243=1038.188,425.768,357.671,174.990,46.105,159.367
C06244=1038.177,425.524,357.720,174.977,46.098,159.364
C06245=1038.166,425.279,357.769,174.964,46.091,159.360
C06246=1038.154,425.034,357.818,174.952,46.084,159.357
C06247=1038.143,424.790,357.867,174.939,46.077,159.353
C06248=1038.131,424.545,357.916,174.926,46.070,159.350
C06249=1038.121,424.299,357.965,174.914,46.064,159.347
C06250=1038.110,424.054,358.014,174.902,46.056,159.343
C06251=1038.098,423.810,358.063,174.889,46.050,159.340
C06252=1038.087,423.564,358.112,174.877,46.043,159.337
C06253=1038.076,423.319,358.161,174.864,46.036,159.334
C06254=1038.065,423.074,358.209,174.852,46.030,159.330
C06255=1038.054,422.829,358.257,174.839,46.023,159.327
C06256=1038.043,422.593,358.304,174.828,46.017,159.324
C06257=1038.032,422.358,358.350,174.816,46.011,159.321
C06258=1038.022,422.124,358.397,174.804,46.004,159.318
C06259=1038.011,421.888,358.443,174.792,45.998,159.315
C06260=1037.999,421.653,358.489,174.781,45.992,159.312
C06261=1037.989,421.419,358.535,174.770,45.985,159.309
C06262=1037.978,421.184,358.582,174.757,45.980,159.306
C06263=1037.968,420.948,358.628,174.746,45.973,159.303
C06264=1037.957,420.704,358.676,174.734,45.967,159.299
C06265=1037.946,420.458,358.725,174.722,45.960,159.296
C06266=1037.935,420.214,358.773,174.710,45.954,159.293
C06267=1037.925,419.968,358.820,174.699,45.948,159.290
C06268=1037.914,419.722,358.868,174.687,45.941,159.287
C06269=1037.903,419.478,358.916,174.675,45.935,159.284
C06270=1037.892,419.232,358.965,174.663,45.928,159.281
C06271=1037.882,418.987,359.012,174.652,45.922,159.278
C06272=1037.871,418.742,359.060,174.640,45.916,159.275
C06273=1037.860,418.497,359.108,174.628,45.909,159.272
C06274=1037.849,418.251,359.155,174.616,45.903,159.269
C06275=1037.838,418.007,359.203,174.605,45.897,159.266
C06276=1037.828,417.761,359.250,174.594,45.891,159.263
C06277=1037.817,417.516,359.299,174.582,45.885,159.260
C06278=1037.807,417.271,359.346,174.571,45.879,159.257
C06279=1037.795,417.025,359.393,174.559,45.872,159.254
C06280=1037.785,416.780,359.440,174.547,45.866,159.251
C06281=1037.774,416.535,359.488,174.536,45.860,159.248
C06282=1037.763,416.289,359.535,174.525,45.854,159.245
C06283=1037.753,416.044,359.582,174.513,45.848,159.242
C06284=1037.743,415.799,359.629,174.502,45.842,159.239
C06285=1037.731,415.553,359.676,174.491,45.836,159.236
C06286=1037.721,415.308,359.724,174.480,45.830,159.233
C06287=1037.711,415.063,359.771,174.470,45.824,159.231
C06288=1037.700,414.818,359.817,174.458,45.818,159.228
C06289=1037.690,414.572,359.865,174.447,45.812,159.225
C06290=1037.679,414.327,359.911,174.436,45.806,159.222
C06291=1037.669,414.081,359.958,174.425,45.800,159.219
C06292=1037.658,413.835,360.005,174.414,45.794,159.216
C06293=1037.647,413.590,360.052,174.403,45.789,159.214
C06294=1037.637,413.345,360.098,174.392,45.782,159.211
C06295=1037.627,413.099,360.146,174.381,45.777,159.208
C06296=1037.616,412.854,360.192,174.371,45.771,159.205
C06297=1037.606,412.608,360.239,174.360,45.765,159.203
C06298=1037.596,412.364,360.284,174.349,45.759,159.200
C06299=1037.586,412.118,360.332,174.338,45.754,159.197
C06300=1037.576,411.872,360.378,174.327,45.748,159.194
C06301=1037.565,411.627,360.425,174.317,45.742,159.192
C06302=1037.555,411.381,360.471,174.306,45.736,159.189
C06303=1037.545,411.136,360.517,174.295,45.731,159.186
C06304=1037.535,410.890,360.564,174.284,45.725,159.184
C06305=1037.524,410.644,360.609,174.274,45.719,159.181
C06306=1037.514,410.399,360.655,174.263,45.714,159.178
C06307=1037.503,410.155,360.702,174.254,45.708,159.176
C06308=1037.493,409.909,360.748,174.243,45.703,159.173
C06309=1037.483,409.662,360.793,174.232,45.697,159.170
C06310=1037.472,409.417,360.839,174.222,45.692,159.168
C06311=1037.463,409.172,360.885,174.211,45.686,159.165
C06312=1037.452,408.926,360.931,174.201,45.680,159.162
C06313=1037.442,408.680,360.977,174.191,45.675,159.160
C06314=1037.432,408.435,361.023,174.180,45.670,159.157
C06315=1037.422,408.189,361.069,174.170,45.665,159.155
C06316=1037.412,407.958,361.111,174.161,45.659,159.152
C06317=1037.403,407.728,361.155,174.151,45.654,159.150
C06318=1037.393,407.497,361.198,174.142,45.649,159.148
C06319=1037.384,407.267,361.240,174.132,45.644,159.145
C06320=1037.375,407.035,361.283,174.123,45.639,159.143
C06321=1037.365,406.805,361.326,174.113,45.634,159.140
C06322=1037.356,406.574,361.369,174.104,45.629,159.138
C06323=1037.347,406.343,361.411,174.094,45.624,159.136
C06324=1037.332,405.976,361.480,174.080,45.616,159.132
C06325=1037.317,405.608,361.547,174.065,45.608,159.128
C06326=1037.302,405.241,361.615,174.050,45.600,159.125
C06327=1037.288,404.873,361.683,174.034,45.592,159.121
C06328=1037.278,404.628,361.728,174.025,45.588,159.119
C06329=1037.268,404.383,361.773,174.015,45.582,159.116
C06330=1037.259,404.137,361.819,174.006,45.577,159.114
C06331=1037.249,403.890,361.864,173.995,45.572,159.111
C06332=1037.239,403.645,361.909,173.986,45.566,159.109
C06333=1037.229,403.399,361.953,173.977,45.562,159.106
C06334=1037.220,403.154,361.999,173.966,45.556,159.104
C06335=1037.211,402.908,362.044,173.957,45.551,159.102
C06336=1037.200,402.662,362.089,173.947,45.546,159.099
C06337=1037.190,402.416,362.134,173.938,45.541,159.097
C06338=1037.181,402.171,362.178,173.929,45.536,159.095
C06339=1037.171,401.925,362.223,173.919,45.532,159.092
C06340=1037.162,401.679,362.267,173.909,45.526,159.090
C06341=1037.152,401.434,362.312,173.900,45.521,159.088
C06342=1037.143,401.188,362.356,173.890,45.516,159.085
C06343=1037.133,400.942,362.401,173.881,45.511,159.083
C06344=1037.123,400.697,362.446,173.872,45.506,159.081
C06345=1037.114,400.450,362.490,173.863,45.501,159.078
C06346=1037.104,400.205,362.535,173.852,45.497,159.076
C06347=1037.095,399.959,362.579,173.843,45.492,159.074
C06348=1037.085,399.713,362.624,173.834,45.487,159.072
C06349=1037.075,399.467,362.668,173.825,45.482,159.069
C06350=1037.066,399.221,362.712,173.815,45.478,159.067
C06351=1037.056,398.976,362.756,173.806,45.473,159.065
C06352=1037.046,398.730,362.800,173.797,45.468,159.063
C06353=1037.037,398.484,362.844,173.788,45.463,159.060
C06354=1037.028,398.238,362.888,173.779,45.458,159.058
C06355=1037.019,397.992,362.932,173.770,45.453,159.056
C06356=1037.008,397.747,362.977,173.760,45.449,159.054
C06357=1036.999,397.501,363.021,173.751,45.444,159.052
C06358=1036.990,397.255,363.064,173.742,45.439,159.049
C06359=1036.980,397.009,363.109,173.733,45.435,159.047
C06360=1036.971,396.763,363.153,173.724,45.430,159.045
C06361=1036.961,396.517,363.196,173.715,45.425,159.043
C06362=1036.952,396.272,363.240,173.706,45.421,159.041
C06363=1036.943,396.026,363.284,173.697,45.416,159.038
C06364=1036.934,395.779,363.327,173.689,45.412,159.036
C06365=1036.925,395.533,363.371,173.680,45.407,159.034
C06366=1036.915,395.288,363.415,173.671,45.402,159.032
C06367=1036.906,395.042,363.458,173.662,45.398,159.030
C06368=1036.896,394.796,363.503,173.653,45.393,159.028
C06369=1036.887,394.549,363.546,173.644,45.389,159.026
C06370=1036.878,394.304,363.589,173.635,45.384,159.024
C06371=1036.869,394.057,363.632,173.627,45.380,159.022
C06372=1036.859,393.812,363.676,173.618,45.375,159.019
C06373=1036.850,393.565,363.719,173.609,45.371,159.017
C06374=1036.841,393.320,363.763,173.600,45.366,159.015
C06375=1036.831,393.074,363.806,173.591,45.362,159.013
C06376=1036.820,392.754,363.862,173.581,45.356,159.011
C06377=1036.808,392.435,363.918,173.569,45.350,159.008
C06378=1036.796,392.115,363.974,173.558,45.345,159.005
C06379=1036.784,391.796,364.030,173.547,45.339,159.003
C06380=1036.775,391.550,364.074,173.539,45.335,159.001
C06381=1036.766,391.304,364.116,173.530,45.331,158.999
C06382=1036.756,391.057,364.160,173.521,45.326,158.997
C06383=1036.747,390.811,364.202,173.513,45.322,158.995
C06384=1036.739,390.565,364.245,173.505,45.317,158.993
C06385=1036.729,390.319,364.288,173.496,45.314,158.991
C06386=1036.720,390.073,364.331,173.487,45.309,158.989
C06387=1036.711,389.827,364.373,173.479,45.305,158.987
C06388=1036.703,389.581,364.416,173.471,45.301,158.985
C06389=1036.693,389.334,364.459,173.462,45.296,158.983
C06390=1036.684,389.088,364.502,173.454,45.293,158.981
C06391=1036.675,388.843,364.545,173.446,45.288,158.979
C06392=1036.666,388.597,364.587,173.438,45.284,158.977
C06393=1036.657,388.350,364.630,173.429,45.280,158.975
C06394=1036.648,388.104,364.672,173.421,45.276,158.973
C06395=1036.639,387.858,364.715,173.413,45.272,158.971
C06396=1036.630,387.612,364.758,173.404,45.267,158.969
C06397=1036.621,387.366,364.799,173.396,45.264,158.968
C06398=1036.612,387.120,364.842,173.389,45.260,158.966
C06399=1036.604,386.873,364.884,173.380,45.256,158.964
C06400=1036.594,386.627,364.927,173.373,45.252,158.962
C06401=1036.585,386.380,364.969,173.364,45.248,158.960
C06402=1036.576,386.135,365.011,173.355,45.243,158.958
C06403=1036.567,385.888,365.053,173.348,45.239,158.956
C06404=1036.558,385.642,365.094,173.340,45.235,158.955
C06405=1036.549,385.396,365.137,173.331,45.232,158.953
C06406=1036.540,385.150,365.179,173.324,45.228,158.951
C06407=1036.531,384.903,365.221,173.315,45.224,158.949
C06408=1036.522,384.657,365.263,173.308,45.220,158.947
C06409=1036.513,384.411,365.305,173.300,45.216,158.946
C06410=1036.504,384.165,365.347,173.292,45.212,158.944
C06411=1036.496,383.918,365.389,173.284,45.208,158.942
C06412=1036.487,383.672,365.431,173.276,45.204,158.940
C06413=1036.478,383.426,365.473,173.268,45.200,158.938
C06414=1036.469,383.180,365.515,173.261,45.197,158.937
C06415=1036.461,382.934,365.556,173.252,45.193,158.935
C06416=1036.452,382.688,365.598,173.245,45.189,158.933
C06417=1036.443,382.441,365.640,173.237,45.186,158.931
C06418=1036.435,382.194,365.682,173.229,45.182,158.929
C06419=1036.426,381.948,365.724,173.221,45.178,158.928
C06420=1036.417,381.702,365.765,173.214,45.174,158.926
C06421=1036.409,381.455,365.806,173.206,45.170,158.924
C06422=1036.400,381.209,365.848,173.198,45.167,158.923
C06423=1036.391,380.963,365.890,173.190,45.163,158.921
C06424=1036.383,380.717,365.931,173.182,45.159,158.919
C06425=1036.374,380.471,365.973,173.175,45.155,158.917
C06426=1036.366,380.223,366.014,173.168,45.152,158.916
C06427=1036.357,379.977,366.056,173.159,45.148,158.914
C06428=1036.348,379.731,366.097,173.152,45.144,158.912
C06429=1036.340,379.484,366.138,173.145,45.141,158.911
C06430=1036.331,379.239,366.180,173.137,45.137,158.909
C06431=1036.323,378.992,366.221,173.129,45.133,158.907
C06432=1036.309,378.586,366.290,173.117,45.127,158.904
C06433=1036.295,378.178,366.358,173.105,45.121,158.902
C06434=1036.281,377.772,366.426,173.093,45.116,158.899
C06435=1036.266,377.364,366.493,173.080,45.110,158.896
C06436=1036.258,377.117,366.534,173.073,45.106,158.894
C06437=1036.249,376.872,366.575,173.066,45.103,158.893
C06438=1036.240,376.625,366.616,173.057,45.099,158.891
C06439=1036.232,376.379,366.656,173.050,45.096,158.890
C06440=1036.223,376.132,366.697,173.043,45.093,158.888
C06441=1036.215,375.885,366.738,173.036,45.089,158.887
C06442=1036.206,375.639,366.779,173.029,45.086,158.885
C06443=1036.198,375.393,366.820,173.021,45.082,158.883
C06444=1036.189,375.146,366.861,173.014,45.079,158.882
C06445=1036.181,374.900,366.901,173.007,45.075,158.880
C06446=1036.172,374.654,366.941,173.000,45.072,158.879
C06447=1036.164,374.407,366.982,172.993,45.069,158.877
C06448=1036.156,374.161,367.023,172.984,45.065,158.875
C06449=1036.147,373.914,367.064,172.978,45.062,158.874
C06450=1036.138,373.668,367.104,172.970,45.059,158.872
C06451=1036.130,373.421,367.144,172.963,45.055,158.871
C06452=1036.122,373.174,367.185,172.956,45.052,158.869
C06453=1036.114,372.928,367.226,172.949,45.049,158.868
C06454=1036.106,372.681,367.266,172.942,45.045,158.866
C06455=1036.096,372.435,367.307,172.935,45.042,158.865
C06456=1036.089,372.188,367.347,172.928,45.039,158.863
C06457=1036.081,371.941,367.387,172.921,45.036,158.861
C06458=1036.073,371.695,367.428,172.913,45.032,158.860
C06459=1036.064,371.448,367.468,172.906,45.029,158.858
C06460=1036.056,371.201,367.508,172.899,45.026,158.857
C06461=1036.048,370.955,367.549,172.892,45.023,158.855
C06462=1036.040,370.708,367.589,172.885,45.020,158.854
C06463=1036.031,370.462,367.629,172.878,45.016,158.852
C06464=1036.023,370.215,367.669,172.871,45.013,158.851
C06465=1036.015,369.968,367.710,172.864,45.010,158.849
C06466=1036.006,369.722,367.749,172.857,45.006,158.848
C06467=1035.998,369.476,367.790,172.850,45.003,158.846
C06468=1035.990,369.229,367.829,172.844,45.000,158.845
C06469=1035.982,368.982,367.869,172.837,44.997,158.844
C06470=1035.973,368.736,367.909,172.830,44.994,158.842
C06471=1035.964,368.489,367.949,172.823,44.991,158.841
C06472=1035.956,368.242,367.989,172.816,44.988,158.839
C06473=1035.948,367.995,368.028,172.809,44.985,158.838
C06474=1035.940,367.748,368.068,172.802,44.982,158.836
C06475=1035.932,367.502,368.108,172.796,44.979,158.835
C06476=1035.923,367.256,368.147,172.790,44.976,158.834
C06477=1035.915,367.009,368.187,172.783,44.973,158.832
C06478=1035.907,366.762,368.226,172.776,44.970,158.831
C06479=1035.899,366.515,368.266,172.769,44.967,158.829
C06480=1035.891,366.269,368.306,172.762,44.964,158.828
C06481=1035.883,366.022,368.346,172.755,44.961,158.826
C06482=1035.875,365.775,368.385,172.748,44.958,158.825
C06483=1035.866,365.529,368.424,172.742,44.955,158.824
C06484=1035.858,365.282,368.464,172.735,44.953,158.822
C06485=1035.850,365.035,368.503,172.728,44.950,158.821
C06486=1035.842,364.788,368.543,172.722,44.946,158.819
C06487=1035.834,364.541,368.582,172.715,44.943,158.818
C06488=1035.821,364.155,368.644,172.705,44.939,158.816
C06489=1035.809,363.768,368.705,172.695,44.934,158.814
C06490=1035.796,363.383,368.767,172.684,44.930,158.812
C06491=1035.784,362.996,368.828,172.675,44.926,158.810
C06492=1035.776,362.749,368.868,172.668,44.923,158.808
C06493=1035.768,362.503,368.907,172.661,44.920,158.807
C06494=1035.760,362.255,368.946,172.654,44.917,158.806
C06495=1035.752,362.009,368.985,172.648,44.914,158.804
C06496=1035.744,361.762,369.024,172.642,44.911,158.803
C06497=1035.736,361.515,369.064,172.635,44.908,158.802
C06498=1035.728,361.268,369.103,172.628,44.906,158.800
C06499=1035.720,361.022,369.141,172.623,44.903,158.799
C06500=1035.712,360.775,369.180,172.616,44.900,158.798
C06501=1035.704,360.528,369.219,172.609,44.898,158.796
C06502=1035.696,360.281,369.258,172.603,44.895,158.795
C06503=1035.689,360.034,369.297,172.597,44.892,158.794
C06504=1035.680,359.787,369.336,172.590,44.890,158.792
C06505=1035.672,359.540,369.375,172.584,44.887,158.791
C06506=1035.665,359.294,369.413,172.577,44.884,158.790
C06507=1035.657,359.047,369.452,172.571,44.881,158.789
C06508=1035.648,358.800,369.491,172.565,44.879,158.787
C06509=1035.641,358.553,369.529,172.558,44.877,158.786
C06510=1035.632,358.306,369.568,172.553,44.874,158.785
C06511=1035.624,358.059,369.606,172.546,44.871,158.784
C06512=1035.617,357.812,369.645,172.539,44.868,158.782
C06513=1035.609,357.565,369.683,172.534,44.866,158.781
C06514=1035.601,357.319,369.722,172.527,44.863,158.780
C06515=1035.593,357.072,369.760,172.520,44.861,158.779
C06516=1035.585,356.825,369.798,172.515,44.858,158.777
C06517=1035.577,356.578,369.837,172.508,44.856,158.776
C06518=1035.569,356.331,369.876,172.503,44.853,158.775
C06519=1035.562,356.084,369.914,172.496,44.850,158.774
C06520=1035.554,355.837,369.953,172.489,44.848,158.772
C06521=1035.546,355.590,369.991,172.484,44.845,158.771
C06522=1035.538,355.343,370.029,172.477,44.843,158.770
C06523=1035.530,355.097,370.068,172.472,44.841,158.769
C06524=1035.522,354.849,370.105,172.465,44.838,158.768
C06525=1035.515,354.602,370.144,172.459,44.836,158.766
C06526=1035.506,354.355,370.182,172.453,44.833,158.765
C06527=1035.499,354.109,370.221,172.447,44.831,158.764
C06528=1035.491,353.862,370.257,172.441,44.828,158.763
C06529=1035.483,353.614,370.296,172.435,44.826,158.762
C06530=1035.475,353.368,370.334,172.429,44.823,158.761
C06531=1035.467,353.120,370.372,172.423,44.821,158.759
C06532=1035.460,352.874,370.410,172.416,44.819,158.758
C06533=1035.453,352.626,370.448,172.411,44.816,158.757
C06534=1035.444,352.380,370.486,172.404,44.814,158.756
C06535=1035.436,352.132,370.524,172.399,44.812,158.755
C06536=1035.429,351.886,370.562,172.392,44.809,158.753
C06537=1035.421,351.638,370.600,172.387,44.806,158.752
C06538=1035.414,351.392,370.638,172.380,44.804,158.751
C06539=1035.406,351.144,370.675,172.375,44.802,158.750
C06540=1035.398,350.897,370.714,172.369,44.800,158.749
C06541=1035.390,350.650,370.751,172.363,44.797,158.748
C06542=1035.383,350.404,370.789,172.358,44.795,158.747
C06543=1035.375,350.157,370.827,172.351,44.793,158.745
C06544=1035.364,349.776,370.884,172.342,44.789,158.744
C06545=1035.352,349.396,370.943,172.333,44.785,158.742
C06546=1035.340,349.015,371.001,172.325,44.782,158.740
C06547=1035.328,348.636,371.058,172.315,44.779,158.739
C06548=1035.320,348.388,371.096,172.309,44.776,158.737
C06549=1035.312,348.141,371.133,172.304,44.774,158.736
C06550=1035.305,347.894,371.171,172.297,44.772,158.735
C06551=1035.297,347.647,371.208,172.292,44.770,158.734
C06552=1035.290,347.400,371.245,172.286,44.767,158.733
C06553=1035.282,347.153,371.283,172.280,44.765,158.732
C06554=1035.274,346.905,371.320,172.275,44.763,158.731
C06555=1035.267,346.658,371.358,172.268,44.761,158.730
C06556=1035.259,346.411,371.395,172.263,44.759,158.729
C06557=1035.251,346.164,371.432,172.258,44.757,158.728
C06558=1035.243,345.917,371.469,172.251,44.755,158.727
C06559=1035.236,345.670,371.507,172.246,44.753,158.726
C06560=1035.229,345.423,371.544,172.241,44.750,158.725
C06561=1035.221,345.176,371.580,172.234,44.749,158.724
C06562=1035.214,344.929,371.618,172.229,44.746,158.722
C06563=1035.206,344.682,371.655,172.224,44.744,158.721
C06564=1035.199,344.435,371.692,172.217,44.742,158.720
C06565=1035.191,344.188,371.729,172.212,44.740,158.719
C06566=1035.184,343.940,371.766,172.207,44.738,158.718
C06567=1035.176,343.693,371.803,172.200,44.736,158.717
C06568=1035.169,343.446,371.840,172.195,44.734,158.716
C06569=1035.161,343.199,371.877,172.190,44.732,158.715
C06570=1035.154,342.951,371.914,172.184,44.730,158.714
C06571=1035.146,342.705,371.951,172.178,44.728,158.713
C06572=1035.138,342.457,371.987,172.173,44.726,158.712
C06573=1035.131,342.210,372.025,172.168,44.724,158.711
C06574=1035.123,341.963,372.061,172.161,44.722,158.710
C06575=1035.116,341.716,372.099,172.156,44.720,158.709
C06576=1035.108,341.469,372.136,172.151,44.717,158.708
C06577=1035.101,341.221,372.172,172.146,44.716,158.707
C06578=1035.093,340.973,372.209,172.139,44.714,158.706
C06579=1035.085,340.727,372.246,172.134,44.712,158.705
C06580=1035.079,340.480,372.282,172.129,44.710,158.704
C06581=1035.071,340.233,372.319,172.124,44.708,158.703
C06582=1035.063,339.985,372.355,172.117,44.706,158.702
C06583=1035.056,339.738,372.391,172.112,44.704,158.701
C06584=1035.048,339.491,372.428,172.107,44.702,158.700
C06585=1035.041,339.243,372.465,172.102,44.700,158.699
C06586=1035.033,338.996,372.501,172.095,44.698,158.698
C06587=1035.026,338.749,372.537,172.090,44.697,158.697
C06588=1035.018,338.502,372.573,172.085,44.695,158.696
C06589=1035.010,338.255,372.610,172.080,44.693,158.695
C06590=1035.003,338.007,372.647,172.074,44.691,158.694
C06591=1034.996,337.760,372.683,172.068,44.689,158.693
C06592=1034.989,337.513,372.719,172.063,44.688,158.692
C06593=1034.981,337.265,372.755,172.058,44.685,158.691
C06594=1034.973,337.018,372.792,172.053,44.684,158.691
C06595=1034.966,336.770,372.828,172.048,44.682,158.690
C06596=1034.959,336.524,372.865,172.042,44.680,158.689
C06597=1034.951,336.277,372.901,172.036,44.678,158.688
C06598=1034.944,336.029,372.937,172.031,44.677,158.687
C06599=1034.936,335.783,372.973,172.026,44.675,158.686
C06600=1034.925,335.398,373.030,172.018,44.672,158.684
C06601=1034.914,335.014,373.085,172.010,44.669,158.683
C06602=1034.903,334.630,373.142,172.002,44.667,158.682
C06603=1034.891,334.247,373.198,171.993,44.664,158.680
C06604=1034.884,334.000,373.234,171.988,44.662,158.679
C06605=1034.877,333.752,373.269,171.983,44.660,158.678
C06606=1034.869,333.505,373.305,171.978,44.659,158.677
C06607=1034.861,333.258,373.341,171.973,44.657,158.677
C06608=1034.854,333.011,373.377,171.968,44.655,158.676
C06609=1034.846,332.763,373.412,171.963,44.654,158.675
C06610=1034.839,332.516,373.448,171.957,44.652,158.674
C06611=1034.832,332.269,373.484,171.952,44.650,158.673
C06612=1034.824,332.021,373.520,171.946,44.649,158.672
C06613=1034.817,331.774,373.556,171.941,44.647,158.671
C06614=1034.810,331.527,373.592,171.936,44.646,158.670
C06615=1034.803,331.279,373.627,171.931,44.644,158.670
C06616=1034.795,331.032,373.663,171.926,44.642,158.669
C06617=1034.788,330.784,373.698,171.921,44.640,158.668
C06618=1034.781,330.537,373.735,171.916,44.639,158.667
C06619=1034.774,330.290,373.770,171.911,44.637,158.666
C06620=1034.766,330.042,373.806,171.906,44.636,158.665
C06621=1034.759,329.795,373.841,171.901,44.634,158.664
C06622=1034.751,329.548,373.877,171.896,44.633,158.663
C06623=1034.744,329.300,373.912,171.891,44.631,158.663
C06624=1034.737,329.054,373.948,171.885,44.629,158.662
C06625=1034.730,328.805,373.983,171.880,44.628,158.661
C06626=1034.723,328.558,374.018,171.875,44.626,158.660
C06627=1034.715,328.311,374.055,171.870,44.625,158.659
C06628=1034.709,328.063,374.090,171.865,44.623,158.658
C06629=1034.701,327.816,374.125,171.860,44.622,158.657
C06630=1034.694,327.568,374.160,171.855,44.620,158.657
C06631=1034.686,327.322,374.195,171.850,44.619,158.656
C06632=1034.679,327.074,374.230,171.845,44.618,158.655
C06633=1034.671,326.827,374.265,171.840,44.616,158.654
C06634=1034.664,326.579,374.301,171.835,44.614,158.653
C06635=1034.656,326.331,374.335,171.831,44.613,158.653
C06636=1034.649,326.084,374.370,171.826,44.612,158.652
C06637=1034.641,325.836,374.405,171.821,44.610,158.651
C06638=1034.635,325.589,374.440,171.815,44.609,158.650
C06639=1034.626,325.341,374.475,171.811,44.608,158.650
C06640=1034.620,325.094,374.510,171.806,44.606,158.649
C06641=1034.612,324.847,374.545,171.801,44.605,158.648
C06642=1034.605,324.599,374.580,171.796,44.604,158.647
C06643=1034.597,324.352,374.615,171.791,44.602,158.646
C06644=1034.590,324.105,374.649,171.786,44.600,158.645
C06645=1034.583,323.857,374.685,171.781,44.600,158.645
C06646=1034.575,323.610,374.719,171.776,44.598,158.644
C06647=1034.568,323.362,374.755,171.771,44.596,158.643
C06648=1034.561,323.115,374.789,171.766,44.595,158.642
C06649=1034.554,322.868,374.824,171.761,44.594,158.642
C06650=1034.546,322.619,374.858,171.756,44.593,158.641
C06651=1034.539,322.372,374.894,171.751,44.591,158.640
C06652=1034.532,322.125,374.928,171.746,44.590,158.639
C06653=1034.525,321.878,374.963,171.742,44.589,158.639
C06654=1034.517,321.630,374.998,171.738,44.588,158.638
C06655=1034.510,321.382,375.033,171.733,44.586,158.637
C06656=1034.499,320.994,375.087,171.725,44.584,158.636
C06657=1034.488,320.606,375.142,171.718,44.582,158.635
C06658=1034.477,320.218,375.196,171.709,44.580,158.634
C06659=1034.465,319.829,375.250,171.702,44.578,158.632
C06660=1034.458,319.582,375.285,171.698,44.577,158.632
C06661=1034.451,319.334,375.319,171.693,44.575,158.631
C06662=1034.444,319.087,375.354,171.688,44.574,158.630
C06663=1034.437,318.840,375.388,171.683,44.573,158.629
C06664=1034.430,318.592,375.422,171.679,44.572,158.629
C06665=1034.423,318.345,375.457,171.674,44.571,158.628
C06666=1034.416,318.097,375.491,171.669,44.569,158.627
C06667=1034.409,317.850,375.526,171.665,44.568,158.626
C06668=1034.402,317.602,375.560,171.660,44.566,158.626
C06669=1034.395,317.354,375.595,171.655,44.565,158.625
C06670=1034.388,317.107,375.629,171.650,44.564,158.624
C06671=1034.380,316.860,375.664,171.645,44.563,158.623
C06672=1034.374,316.612,375.698,171.642,44.562,158.623
C06673=1034.366,316.365,375.733,171.637,44.561,158.622
C06674=1034.360,316.117,375.767,171.632,44.560,158.621
C06675=1034.353,315.869,375.801,171.627,44.558,158.621
C06676=1034.346,315.622,375.836,171.622,44.557,158.620
C06677=1034.339,315.374,375.870,171.618,44.556,158.619
C06678=1034.331,315.126,375.904,171.613,44.554,158.618
C06679=1034.325,314.879,375.939,171.609,44.553,158.618
C06680=1034.318,314.631,375.973,171.604,44.552,158.617
C06681=1034.311,314.383,376.007,171.600,44.551,158.616
C06682=1034.304,314.137,376.041,171.595,44.549,158.616
C06683=1034.297,313.889,376.075,171.590,44.548,158.615
C06684=1034.290,313.641,376.109,171.585,44.547,158.614
C06685=1034.283,313.394,376.143,171.582,44.546,158.614
C06686=1034.277,313.146,376.178,171.577,44.545,158.613
C06687=1034.270,312.899,376.212,171.572,44.544,158.612
C06688=1034.263,312.652,376.246,171.568,44.542,158.611
C06689=1034.256,312.404,376.280,171.563,44.541,158.611
C06690=1034.249,312.156,376.314,171.559,44.541,158.610
C06691=1034.242,311.909,376.349,171.554,44.540,158.609
C06692=1034.236,311.662,376.383,171.550,44.538,158.609
C06693=1034.229,311.414,376.416,171.545,44.537,158.608
C06694=1034.221,311.166,376.450,171.540,44.536,158.607
C06695=1034.214,310.919,376.484,171.537,44.535,158.607
C06696=1034.206,310.671,376.517,171.532,44.534,158.606
C06697=1034.199,310.423,376.550,171.527,44.533,158.605
C06698=1034.193,310.176,376.584,171.522,44.532,158.605
C06699=1034.185,309.928,376.618,171.519,44.532,158.604
C06700=1034.178,309.681,376.651,171.514,44.531,158.604
C06701=1034.171,309.433,376.684,171.509,44.530,158.603
C06702=1034.163,309.185,376.718,171.504,44.529,158.602
C06703=1034.157,308.938,376.751,171.501,44.527,158.602
C06704=1034.150,308.690,376.785,171.496,44.526,158.601
C06705=1034.142,308.443,376.819,171.491,44.526,158.600
C06706=1034.135,308.195,376.851,171.487,44.525,158.600
C06707=1034.128,307.948,376.885,171.483,44.524,158.599
C06708=1034.121,307.700,376.919,171.478,44.523,158.598
C06709=1034.114,307.452,376.952,171.473,44.523,158.598
C06710=1034.106,307.204,376.985,171.470,44.521,158.597
C06711=1034.100,306.957,377.018,171.465,44.520,158.597
C06712=1034.089,306.573,377.070,171.458,44.519,158.596
C06713=1034.078,306.190,377.122,171.452,44.518,158.595
C06714=1034.067,305.807,377.172,171.445,44.516,158.594
C06715=1034.056,305.423,377.225,171.437,44.515,158.593
C06716=1034.049,305.176,377.258,171.434,44.514,158.592
C06717=1034.042,304.928,377.291,171.429,44.513,158.592
C06718=1034.035,304.680,377.325,171.424,44.512,158.591
C06719=1034.028,304.433,377.357,171.421,44.512,158.590
C06720=1034.021,304.185,377.391,171.416,44.511,158.590
C06721=1034.014,303.938,377.423,171.411,44.510,158.589
C06722=1034.007,303.689,377.456,171.408,44.509,158.589
C06723=1034.000,303.442,377.490,171.403,44.508,158.588
C06724=1033.994,303.194,377.523,171.400,44.507,158.587
C06725=1033.986,302.946,377.557,171.395,44.506,158.587
C06726=1033.979,302.699,377.589,171.390,44.505,158.586
C06727=1033.973,302.451,377.622,171.386,44.505,158.586
C06728=1033.966,302.204,377.655,171.382,44.504,158.585
C06729=1033.959,301.956,377.689,171.378,44.503,158.584
C06730=1033.952,301.708,377.721,171.373,44.502,158.584
C06731=1033.945,301.461,377.755,171.369,44.501,158.583
C06732=1033.938,301.213,377.787,171.365,44.501,158.583
C06733=1033.931,300.965,377.820,171.360,44.500,158.582
C06734=1033.924,300.718,377.853,171.357,44.499,158.582
C06735=1033.917,300.470,377.886,171.352,44.498,158.581
C06736=1033.911,300.222,377.919,171.348,44.497,158.580
C06737=1033.903,299.974,377.952,171.344,44.496,158.580
C06738=1033.897,299.727,377.984,171.339,44.496,158.579
C06739=1033.890,299.479,378.018,171.335,44.495,158.579
C06740=1033.884,299.231,378.051,171.331,44.494,158.578
C06741=1033.877,298.984,378.083,171.327,44.493,158.577
C06742=1033.870,298.736,378.116,171.323,44.493,158.577
C06743=1033.863,298.488,378.149,171.319,44.492,158.576
C06744=1033.857,298.240,378.182,171.314,44.491,158.576
C06745=1033.850,297.993,378.214,171.311,44.491,158.575
C06746=1033.843,297.746,378.248,171.306,44.490,158.575
C06747=1033.836,297.497,378.281,171.302,44.489,158.574
C06748=1033.829,297.250,378.313,171.298,44.488,158.573
C06749=1033.823,297.002,378.346,171.294,44.487,158.573
C06750=1033.816,296.754,378.379,171.289,44.486,158.572
C06751=1033.810,296.507,378.412,171.286,44.486,158.572
C06752=1033.802,296.259,378.444,171.281,44.485,158.571
C06753=1033.796,296.011,378.477,171.278,44.484,158.571
C06754=1033.789,295.763,378.510,171.273,44.484,158.570
C06755=1033.782,295.516,378.542,171.269,44.483,158.570
C06756=1033.775,295.268,378.575,171.265,44.482,158.569
C06757=1033.769,295.020,378.608,171.261,44.482,158.569
C06758=1033.763,294.772,378.640,171.257,44.480,158.568
C06759=1033.756,294.525,378.672,171.253,44.480,158.567
C06760=1033.748,294.277,378.704,171.249,44.479,158.567
C06761=1033.742,294.029,378.737,171.245,44.479,158.566
C06762=1033.735,293.782,378.769,171.241,44.478,158.566
C06763=1033.729,293.533,378.801,171.237,44.477,158.565
C06764=1033.721,293.286,378.834,171.233,44.477,158.565
C06765=1033.714,293.038,378.866,171.228,44.476,158.564
C06766=1033.708,292.789,378.898,171.225,44.476,158.564
C06767=1033.701,292.542,378.930,171.220,44.475,158.563
C06768=1033.691,292.176,378.977,171.215,44.475,158.563
C06769=1033.680,291.809,379.025,171.209,44.474,158.562
C06770=1033.670,291.443,379.072,171.203,44.473,158.561
C06771=1033.661,291.076,379.120,171.197,44.472,158.560
C06772=1033.653,290.828,379.152,171.192,44.471,158.560
C06773=1033.646,290.581,379.185,171.189,44.471,158.559
C06774=1033.640,290.333,379.217,171.184,44.470,158.559
C06775=1033.633,290.085,379.249,171.181,44.470,158.558
C06776=1033.626,289.837,379.280,171.176,44.469,158.558
C06777=1033.619,289.589,379.312,171.173,44.469,158.557
C06778=1033.613,289.341,379.345,171.169,44.468,158.557
C06779=1033.606,289.093,379.376,171.165,44.468,158.556
C06780=1033.599,288.846,379.408,171.161,44.467,158.556
C06781=1033.592,288.598,379.440,171.157,44.466,158.555
C06782=1033.585,288.350,379.472,171.153,44.466,158.555
C06783=1033.579,288.102,379.504,171.150,44.465,158.555
C06784=1033.572,287.854,379.536,171.145,44.465,158.554
C06785=1033.565,287.607,379.568,171.142,44.464,158.554
C06786=1033.558,287.359,379.599,171.137,44.464,158.553
C06787=1033.551,287.111,379.631,171.134,44.463,158.553
C06788=1033.544,286.863,379.663,171.130,44.463,158.552
C06789=1033.538,286.615,379.695,171.126,44.463,158.552
C06790=1033.531,286.367,379.727,171.122,44.462,158.551
C06791=1033.524,286.119,379.758,171.118,44.462,158.551
C06792=1033.518,285.871,379.790,171.114,44.461,158.550
C06793=1033.511,285.624,379.822,171.111,44.461,158.550
C06794=1033.504,285.376,379.853,171.106,44.460,158.549
C06795=1033.497,285.128,379.885,171.103,44.460,158.549
C06796=1033.490,284.880,379.915,171.098,44.460,158.549
C06797=1033.482,284.632,379.947,171.095,44.459,158.548
C06798=1033.476,284.384,379.979,171.091,44.459,158.548
C06799=1033.469,284.136,380.010,171.087,44.458,158.547
C06800=1033.462,283.888,380.041,171.084,44.458,158.547
C06801=1033.455,283.640,380.073,171.080,44.458,158.546
C06802=1033.449,283.392,380.104,171.075,44.457,158.546
C06803=1033.442,283.145,380.136,171.072,44.457,158.545
C06804=1033.435,282.897,380.168,171.068,44.457,158.545
C06805=1033.428,282.649,380.199,171.064,44.456,158.545
C06806=1033.422,282.401,380.231,171.061,44.456,158.544
C06807=1033.415,282.153,380.262,171.056,44.455,158.544
C06808=1033.408,281.905,380.293,171.053,44.455,158.543
C06809=1033.402,281.657,380.324,171.049,44.455,158.543
C06810=1033.395,281.409,380.356,171.045,44.454,158.542
C06811=1033.388,281.161,380.387,171.041,44.454,158.542
C06812=1033.381,280.913,380.419,171.038,44.454,158.541
C06813=1033.375,280.665,380.450,171.033,44.453,158.541
C06814=1033.367,280.418,380.481,171.030,44.453,158.540
C06815=1033.361,280.170,380.512,171.027,44.453,158.540
C06816=1033.354,279.922,380.544,171.023,44.452,158.540
C06817=1033.347,279.674,380.575,171.019,44.452,158.539
C06818=1033.341,279.426,380.606,171.015,44.452,158.539
C06819=1033.334,279.178,380.637,171.012,44.451,158.538
C06820=1033.327,278.930,380.669,171.007,44.451,158.538
C06821=1033.321,278.682,380.700,171.004,44.451,158.538
C06822=1033.314,278.435,380.731,171.000,44.450,158.537
C06823=1033.308,278.186,380.762,170.997,44.449,158.537
C06824=1033.298,277.832,380.807,170.991,44.449,158.536
C06825=1033.288,277.477,380.851,170.986,44.449,158.536
C06826=1033.279,277.123,380.895,170.980,44.449,158.535
C06827=1033.269,276.768,380.939,170.976,44.448,158.534
C06828=1033.262,276.520,380.971,170.971,44.448,158.534
C06829=1033.255,276.271,381.001,170.968,44.448,158.534
C06830=1033.248,276.025,381.032,170.964,44.447,158.533
C06831=1033.242,275.777,381.063,170.961,44.447,158.533
C06832=1033.235,275.528,381.094,170.957,44.447,158.532
C06833=1033.228,275.281,381.125,170.953,44.447,158.532
C06834=1033.221,275.032,381.156,170.950,44.446,158.532
C06835=1033.215,274.784,381.187,170.947,44.446,158.531
C06836=1033.208,274.536,381.217,170.942,44.446,158.531
C06837=1033.201,274.289,381.248,170.939,44.446,158.531
C06838=1033.195,274.040,381.279,170.935,44.445,158.530
C06839=1033.188,273.793,381.310,170.932,44.445,158.530
C06840=1033.181,273.544,381.340,170.927,44.445,158.529
C06841=1033.174,273.297,381.371,170.924,44.445,158.529
C06842=1033.167,273.048,381.402,170.921,44.445,158.529
C06843=1033.161,272.800,381.432,170.917,44.444,158.528
C06844=1033.154,272.553,381.463,170.913,44.445,158.528
C06845=1033.148,272.304,381.494,170.910,44.444,158.527
C06846=1033.140,272.056,381.524,170.906,44.444,158.527
C06847=1033.134,271.809,381.555,170.903,44.444,158.527
C06848=1033.128,271.560,381.586,170.900,44.443,158.526
C06849=1033.121,271.312,381.616,170.895,44.443,158.526
C06850=1033.114,271.064,381.647,170.892,44.443,158.525
C06851=1033.107,270.816,381.677,170.888,44.443,158.525
C06852=1033.101,270.568,381.708,170.885,44.443,158.525
C06853=1033.094,270.320,381.739,170.881,44.442,158.524
C06854=1033.087,270.072,381.769,170.877,44.442,158.524
C06855=1033.081,269.824,381.799,170.874,44.442,158.524
C06856=1033.073,269.576,381.829,170.871,44.442,158.523
C06857=1033.067,269.328,381.860,170.867,44.442,158.523
C06858=1033.060,269.079,381.890,170.863,44.442,158.523
C06859=1033.054,268.832,381.921,170.860,44.442,158.522
C06860=1033.047,268.584,381.951,170.856,44.442,158.522
C06861=1033.040,268.335,381.982,170.853,44.441,158.522
C06862=1033.033,268.087,382.012,170.850,44.441,158.521
C06863=1033.026,267.840,382.042,170.846,44.441,158.521
C06864=1033.020,267.591,382.073,170.842,44.442,158.521
C06865=1033.013,267.343,382.103,170.839,44.441,158.520
C06866=1033.007,267.095,382.133,170.835,44.441,158.520
C06867=1033.000,266.847,382.163,170.832,44.441,158.519
C06868=1032.993,266.599,382.193,170.829,44.441,158.519
C06869=1032.987,266.351,382.224,170.824,44.441,158.519
C06870=1032.980,266.103,382.254,170.821,44.441,158.518
C06871=1032.973,265.854,382.284,170.818,44.441,158.518
C06872=1032.966,265.607,382.314,170.814,44.441,158.518
C06873=1032.960,265.358,382.344,170.811,44.441,158.517
C06874=1032.952,265.110,382.374,170.808,44.441,158.517
C06875=1032.946,264.863,382.404,170.804,44.441,158.517
C06876=1032.939,264.615,382.434,170.800,44.441,158.516
C06877=1032.933,264.367,382.465,170.797,44.440,158.516
C06878=1032.926,264.118,382.495,170.793,44.440,158.516
C06879=1032.919,263.870,382.524,170.790,44.440,158.515
C06880=1032.910,263.520,382.567,170.785,44.441,158.515
C06881=1032.901,263.170,382.610,170.780,44.440,158.514
C06882=1032.891,262.820,382.651,170.776,44.440,158.514
C06883=1032.882,262.471,382.694,170.771,44.440,158.514
C06884=1032.875,262.223,382.724,170.767,44.440,158.513
C06885=1032.868,261.975,382.754,170.764,44.440,158.513
C06886=1032.862,261.726,382.784,170.761,44.440,158.513
C06887=1032.855,261.479,382.813,170.757,44.440,158.512
C06888=1032.848,261.230,382.843,170.754,44.440,158.512
C06889=1032.841,260.981,382.873,170.751,44.440,158.512
C06890=1032.835,260.734,382.903,170.747,44.440,158.511
C06891=1032.827,260.485,382.931,170.743,44.440,158.511
C06892=1032.821,260.238,382.961,170.740,44.440,158.511
C06893=1032.814,259.990,382.991,170.737,44.440,158.510
C06894=1032.807,259.742,383.020,170.733,44.440,158.510
C06895=1032.800,259.493,383.051,170.730,44.440,158.510
C06896=1032.793,259.245,383.080,170.727,44.441,158.510
C06897=1032.787,258.997,383.110,170.723,44.441,158.509
C06898=1032.779,258.748,383.138,170.720,44.441,158.509
C06899=1032.773,258.501,383.168,170.716,44.441,158.509
C06900=1032.766,258.252,383.198,170.713,44.441,158.508
C06901=1032.759,258.005,383.227,170.710,44.441,158.508
C06902=1032.752,257.756,383.257,170.706,44.441,158.508
C06903=1032.746,257.508,383.286,170.703,44.442,158.508
C06904=1032.739,257.259,383.316,170.700,44.442,158.507
C06905=1032.732,257.012,383.344,170.696,44.442,158.507
C06906=1032.725,256.763,383.375,170.693,44.442,158.507
C06907=1032.719,256.515,383.404,170.689,44.442,158.506
C06908=1032.711,256.267,383.434,170.686,44.442,158.506
C06909=1032.705,256.019,383.463,170.683,44.442,158.506
C06910=1032.698,255.770,383.492,170.680,44.443,158.506
C06911=1032.691,255.523,383.521,170.676,44.443,158.505
C06912=1032.684,255.274,383.551,170.673,44.443,158.505
C06913=1032.678,255.026,383.580,170.670,44.443,158.505
C06914=1032.671,254.778,383.610,170.667,44.443,158.504
C06915=1032.664,254.530,383.639,170.664,44.443,158.504
C06916=1032.658,254.281,383.668,170.660,44.443,158.504
C06917=1032.651,254.033,383.697,170.657,44.443,158.504
C06918=1032.644,253.785,383.727,170.654,44.443,158.503
C06919=1032.637,253.537,383.756,170.649,44.444,158.503
C06920=1032.631,253.288,383.785,170.646,44.444,158.503
C06921=1032.625,253.040,383.814,170.643,44.444,158.503
C06922=1032.618,252.792,383.844,170.640,44.444,158.502
C06923=1032.611,252.544,383.873,170.637,44.444,158.502
C06924=1032.604,252.295,383.902,170.633,44.444,158.502
C06925=1032.597,252.047,383.931,170.630,44.445,158.502
C06926=1032.591,251.800,383.961,170.627,44.445,158.501
C06927=1032.584,251.551,383.990,170.624,44.445,158.501
C06928=1032.578,251.303,384.019,170.620,44.445,158.501
C06929=1032.571,251.055,384.048,170.617,44.445,158.500
C06930=1032.564,250.806,384.077,170.614,44.445,158.500
C06931=1032.558,250.558,384.106,170.611,44.445,158.500
C06932=1032.551,250.310,384.135,170.608,44.445,158.500
C06933=1032.544,250.062,384.165,170.605,44.446,158.499
C06934=1032.537,249.814,384.194,170.601,44.446,158.499
C06935=1032.531,249.566,384.223,170.598,44.446,158.499
C06936=1032.522,249.214,384.264,170.594,44.446,158.498
C06937=1032.512,248.863,384.305,170.589,44.447,158.498
C06938=1032.504,248.511,384.346,170.585,44.447,158.498
C06939=1032.494,248.160,384.387,170.580,44.447,158.497
C06940=1032.488,247.912,384.416,170.577,44.447,158.497
C06941=1032.481,247.664,384.445,170.574,44.448,158.497
C06942=1032.474,247.415,384.475,170.570,44.448,158.497
C06943=1032.468,247.167,384.503,170.568,44.448,158.496
C06944=1032.461,246.919,384.532,170.565,44.448,158.496
C06945=1032.455,246.671,384.561,170.562,44.448,158.496
C06946=1032.449,246.423,384.590,170.558,44.448,158.496
C06947=1032.442,246.174,384.620,170.555,44.448,158.495
C06948=1032.435,245.926,384.648,170.552,44.449,158.495
C06949=1032.429,245.678,384.677,170.549,44.449,158.495
C06950=1032.422,245.430,384.706,170.546,44.449,158.494
C06951=1032.416,245.182,384.735,170.542,44.449,158.494
C06952=1032.409,244.933,384.765,170.539,44.449,158.494
C06953=1032.402,244.685,384.793,170.536,44.449,158.494
C06954=1032.396,244.436,384.821,170.533,44.450,158.494
C06955=1032.390,244.188,384.850,170.530,44.450,158.493
C06956=1032.383,243.940,384.879,170.526,44.450,158.493
C06957=1032.376,243.692,384.908,170.523,44.451,158.493
C06958=1032.370,243.443,384.936,170.520,44.451,158.492
C06959=1032.363,243.195,384.965,170.517,44.451,158.492
C06960=1032.356,242.947,384.993,170.515,44.451,158.492
C06961=1032.350,242.699,385.022,170.512,44.452,158.492
C06962=1032.343,242.450,385.051,170.508,44.452,158.492
C06963=1032.337,242.202,385.080,170.505,44.452,158.491
C06964=1032.330,241.954,385.108,170.502,44.452,158.491
C06965=1032.324,241.705,385.136,170.499,44.453,158.491
C06966=1032.317,241.457,385.165,170.496,44.453,158.491
C06967=1032.310,241.209,385.194,170.493,44.453,158.490
C06968=1032.304,240.961,385.222,170.489,44.454,158.490
C06969=1032.297,240.712,385.251,170.486,44.454,158.490
C06970=1032.290,240.464,385.279,170.483,44.454,158.490
C06971=1032.284,240.215,385.308,170.480,44.454,158.489
C06972=1032.277,239.968,385.336,170.477,44.455,158.489
C06973=1032.270,239.719,385.364,170.475,44.455,158.489
C06974=1032.263,239.471,385.392,170.472,44.455,158.489
C06975=1032.257,239.223,385.421,170.469,44.456,158.489
C06976=1032.250,238.974,385.449,170.465,44.456,158.488
C06977=1032.243,238.726,385.477,170.462,44.456,158.488
C06978=1032.237,238.477,385.506,170.459,44.457,158.488
C06979=1032.230,238.229,385.534,170.456,44.457,158.488
C06980=1032.223,237.981,385.562,170.453,44.458,158.488
C06981=1032.216,237.733,385.590,170.450,44.458,158.487
C06982=1032.211,237.484,385.618,170.447,44.458,158.487
C06983=1032.204,237.236,385.647,170.443,44.459,158.487
C06984=1032.197,236.988,385.675,170.441,44.459,158.487
C06985=1032.190,236.739,385.703,170.438,44.459,158.487
C06986=1032.183,236.491,385.731,170.435,44.460,158.487
C06987=1032.177,236.242,385.760,170.432,44.460,158.486
C06988=1032.170,235.994,385.787,170.429,44.461,158.486
C06989=1032.163,235.746,385.816,170.426,44.461,158.486
C06990=1032.156,235.497,385.843,170.423,44.461,158.486
C06991=1032.150,235.249,385.871,170.419,44.462,158.485
C06992=1032.140,234.892,385.912,170.415,44.462,158.485
C06993=1032.131,234.535,385.952,170.411,44.463,158.485
C06994=1032.121,234.178,385.993,170.407,44.463,158.485
C06995=1032.111,233.820,386.033,170.403,44.464,158.484
C06996=1032.105,233.572,386.061,170.400,44.465,158.484
C06997=1032.098,233.324,386.090,170.396,44.465,158.484
C06998=1032.092,233.075,386.117,170.393,44.465,158.484
C06999=1032.085,232.827,386.145,170.390,44.466,158.484
C07000=1032.078,232.578,386.173,170.387,44.466,158.483
C07001=1032.072,232.330,386.201,170.385,44.466,158.483
C07002=1032.066,232.082,386.230,170.382,44.467,158.483
C07003=1032.059,231.833,386.257,170.379,44.467,158.483
C07004=1032.052,231.585,386.285,170.376,44.467,158.483
C07005=1032.045,231.337,386.313,170.373,44.468,158.482
C07006=1032.039,231.088,386.341,170.370,44.469,158.482
C07007=1032.032,230.840,386.368,170.367,44.468,158.482
C07008=1032.025,230.591,386.396,170.364,44.469,158.482
C07009=1032.018,230.343,386.424,170.361,44.470,158.482
C07010=1032.012,230.095,386.452,170.358,44.470,158.482
C07011=1032.005,229.847,386.480,170.355,44.470,158.481
C07012=1031.999,229.599,386.507,170.352,44.471,158.481
C07013=1031.992,229.350,386.535,170.350,44.471,158.481
C07014=1031.986,229.102,386.563,170.347,44.472,158.481
C07015=1031.979,228.853,386.590,170.344,44.472,158.481
C07016=1031.972,228.605,386.618,170.341,44.473,158.480
C07017=1031.966,228.357,386.646,170.338,44.473,158.480
C07018=1031.959,228.108,386.674,170.335,44.474,158.480
C07019=1031.953,227.859,386.702,170.333,44.474,158.480
C07020=1031.946,227.611,386.729,170.329,44.474,158.480
C07021=1031.939,227.363,386.757,170.326,44.475,158.480
C07022=1031.932,227.114,386.784,170.323,44.476,158.479
C07023=1031.926,226.865,386.812,170.320,44.476,158.479
C07024=1031.919,226.617,386.839,170.318,44.477,158.479
C07025=1031.912,226.369,386.866,170.315,44.477,158.479
C07026=1031.906,226.121,386.894,170.312,44.478,158.479
C07027=1031.899,225.873,386.922,170.309,44.478,158.479
C07028=1031.892,225.624,386.949,170.306,44.479,158.479
C07029=1031.885,225.375,386.976,170.303,44.480,158.478
C07030=1031.878,225.127,387.003,170.301,44.480,158.478
C07031=1031.872,224.878,387.031,170.298,44.480,158.478
C07032=1031.865,224.630,387.059,170.295,44.481,158.478
C07033=1031.859,224.381,387.086,170.292,44.481,158.478
C07034=1031.852,224.134,387.113,170.289,44.482,158.478
C07035=1031.845,223.885,387.140,170.286,44.482,158.477
C07036=1031.839,223.637,387.168,170.283,44.483,158.477
C07037=1031.832,223.388,387.196,170.280,44.484,158.477
C07038=1031.825,223.139,387.223,170.277,44.484,158.477
C07039=1031.818,222.891,387.250,170.274,44.485,158.477
C07040=1031.812,222.643,387.277,170.272,44.485,158.477
C07041=1031.806,222.394,387.304,170.269,44.486,158.477
C07042=1031.799,222.146,387.332,170.266,44.487,158.476
C07043=1031.792,221.898,387.359,170.263,44.487,158.476
C07044=1031.785,221.649,387.386,170.261,44.487,158.476
C07045=1031.778,221.400,387.414,170.258,44.488,158.476
C07046=1031.772,221.152,387.441,170.255,44.488,158.476
C07047=1031.766,220.903,387.468,170.252,44.489,158.476
C07048=1031.756,220.539,387.508,170.248,44.490,158.475
C07049=1031.746,220.175,387.548,170.244,44.491,158.475
C07050=1031.737,219.810,387.589,170.240,44.491,158.475
C07051=1031.727,219.445,387.628,170.236,44.492,158.475
C07052=1031.720,219.197,387.655,170.233,44.493,158.475
C07053=1031.713,218.948,387.682,170.231,44.493,158.475
C07054=1031.706,218.699,387.709,170.228,44.494,158.474
C07055=1031.700,218.450,387.736,170.224,44.495,158.474
C07056=1031.693,218.203,387.763,170.221,44.495,158.474
C07057=1031.686,217.954,387.790,170.219,44.496,158.474
C07058=1031.679,217.706,387.817,170.216,44.496,158.474
C07059=1031.673,217.457,387.844,170.213,44.497,158.474
C07060=1031.666,217.209,387.870,170.210,44.498,158.474
C07061=1031.660,216.960,387.898,170.209,44.499,158.474
C07062=1031.652,216.711,387.925,170.205,44.499,158.473
C07063=1031.646,216.463,387.952,170.202,44.500,158.473
C07064=1031.639,216.215,387.978,170.199,44.500,158.473
C07065=1031.633,215.966,388.005,170.197,44.501,158.473
C07066=1031.625,215.718,388.033,170.194,44.501,158.473
C07067=1031.619,215.469,388.060,170.191,44.502,158.473
C07068=1031.613,215.221,388.086,170.188,44.503,158.473
C07069=1031.606,214.972,388.113,170.186,44.503,158.472
C07070=1031.599,214.723,388.140,170.183,44.504,158.472
C07071=1031.593,214.476,388.167,170.180,44.504,158.472
C07072=1031.586,214.227,388.194,170.178,44.505,158.472
C07073=1031.579,213.978,388.221,170.175,44.506,158.472
C07074=1031.573,213.730,388.247,170.172,44.507,158.472
C07075=1031.566,213.481,388.274,170.169,44.507,158.472
C07076=1031.559,213.233,388.301,170.167,44.508,158.472
C07077=1031.552,212.985,388.327,170.164,44.508,158.472
C07078=1031.546,212.736,388.355,170.161,44.509,158.471
C07079=1031.539,212.487,388.381,170.159,44.509,158.471
C07080=1031.533,212.239,388.408,170.156,44.510,158.471
C07081=1031.526,211.990,388.434,170.153,44.511,158.471
C07082=1031.519,211.742,388.462,170.151,44.512,158.471
C07083=1031.512,211.494,388.488,170.148,44.512,158.471
C07084=1031.506,211.245,388.515,170.145,44.513,158.471
C07085=1031.500,210.997,388.541,170.143,44.513,158.471
C07086=1031.493,210.748,388.568,170.140,44.514,158.470
C07087=1031.486,210.500,388.595,170.137,44.515,158.470
C07088=1031.479,210.251,388.621,170.134,44.515,158.470
C07089=1031.472,210.003,388.648,170.132,44.516,158.470
C07090=1031.466,209.754,388.675,170.129,44.517,158.470
C07091=1031.459,209.506,388.701,170.126,44.518,158.470
C07092=1031.452,209.257,388.727,170.124,44.518,158.470
C07093=1031.446,209.008,388.754,170.121,44.519,158.470
C07094=1031.439,208.760,388.780,170.118,44.520,158.470
C07095=1031.432,208.511,388.806,170.116,44.520,158.470
C07096=1031.426,208.263,388.833,170.113,44.521,158.469
C07097=1031.419,208.014,388.860,170.110,44.522,158.469
C07098=1031.413,207.766,388.886,170.108,44.523,158.469
C07099=1031.406,207.517,388.912,170.105,44.523,158.469
C07100=1031.399,207.268,388.938,170.102,44.524,158.469
C07101=1031.392,207.020,388.965,170.100,44.524,158.469
C07102=1031.386,206.771,388.992,170.098,44.526,158.469
C07103=1031.379,206.523,389.018,170.095,44.526,158.469
C07104=1031.369,206.164,389.056,170.090,44.527,158.469
C07105=1031.359,205.805,389.094,170.088,44.528,158.469
C07106=1031.350,205.446,389.132,170.084,44.529,158.468
C07107=1031.339,205.088,389.169,170.080,44.531,158.468
C07108=1031.314,204.038,389.275,169.730,44.426,158.414
C07109=1031.307,203.790,389.300,169.727,44.428,158.414
C07110=1031.302,203.541,389.324,169.723,44.430,158.414
C07111=1031.296,203.293,389.350,169.719,44.431,158.414
C07112=1031.290,203.043,389.374,169.715,44.433,158.414
C07113=1031.284,202.795,389.400,169.712,44.434,158.414
C07114=1031.277,202.547,389.424,169.709,44.435,158.414
C07115=1031.272,202.298,389.449,169.705,44.437,158.414
C07116=1031.265,202.049,389.474,169.701,44.438,158.414
C07117=1031.260,201.800,389.498,169.697,44.440,158.414
C07118=1031.254,201.552,389.523,169.694,44.442,158.414
C07119=1031.248,201.302,389.548,169.691,44.443,158.414
C07120=1031.242,201.054,389.573,169.687,44.445,158.414
C07121=1031.236,200.806,389.597,169.683,44.446,158.414
C07122=1031.229,200.557,389.622,169.680,44.448,158.414
C07123=1031.224,200.308,389.647,169.676,44.449,158.413
C07124=1031.217,200.060,389.671,169.673,44.451,158.414
C07125=1031.211,199.811,389.696,169.669,44.452,158.414
C07126=1031.205,199.562,389.720,169.666,44.454,158.414
C07127=1031.198,199.313,389.745,169.662,44.456,158.414
C07128=1031.192,199.065,389.769,169.658,44.457,158.414
C07129=1031.187,198.815,389.794,169.654,44.459,158.414
C07130=1031.180,198.567,389.818,169.652,44.461,158.414
C07131=1031.174,198.318,389.843,169.648,44.462,158.414
C07132=1031.168,198.069,389.867,169.644,44.464,158.414
C07133=1031.162,197.820,389.891,169.641,44.466,158.414
C07134=1031.155,197.573,389.916,169.637,44.467,158.414
C07135=1031.150,197.323,389.940,169.634,44.469,158.414
C07136=1031.143,197.074,389.964,169.630,44.471,158.414
C07137=1031.138,196.826,389.989,169.627,44.472,158.414
C07138=1031.131,196.577,390.013,169.623,44.474,158.414
C07139=1031.125,196.329,390.038,169.619,44.476,158.414
C07140=1031.119,196.080,390.062,169.616,44.477,158.414
C07141=1031.113,195.830,390.086,169.613,44.479,158.414
C07142=1031.107,195.582,390.110,169.609,44.481,158.414
C07143=1031.101,195.334,390.135,169.605,44.483,158.414
C07144=1031.095,195.085,390.159,169.603,44.484,158.414
C07145=1031.089,194.836,390.184,169.599,44.486,158.414
C07146=1031.082,194.587,390.208,169.595,44.488,158.414
C07147=1031.077,194.338,390.232,169.591,44.489,158.414
C07148=1031.070,194.089,390.256,169.589,44.491,158.414
C07149=1031.065,193.841,390.280,169.585,44.493,158.414
C07150=1031.058,193.592,390.304,169.581,44.494,158.414
C07151=1031.053,193.343,390.328,169.578,44.496,158.414
C07152=1031.046,193.095,390.353,169.575,44.497,158.414
C07153=1031.041,192.846,390.377,169.571,44.500,158.414
C07154=1031.034,192.597,390.401,169.567,44.501,158.414
C07155=1031.028,192.349,390.425,169.565,44.503,158.414
C07156=1031.022,192.100,390.450,169.561,44.504,158.414
C07157=1031.016,191.851,390.473,169.557,44.506,158.414
C07158=1031.010,191.602,390.498,169.554,44.508,158.414
C07159=1031.004,191.354,390.522,169.551,44.509,158.414
C07160=1030.998,191.105,390.546,169.547,44.511,158.414
C07161=1030.992,190.856,390.570,169.543,44.513,158.414
C07162=1030.986,190.607,390.595,169.541,44.515,158.414
C07163=1030.980,190.359,390.618,169.537,44.516,158.414
C07164=1030.974,190.109,390.643,169.533,44.518,158.414
C07165=1030.969,189.861,390.666,169.531,44.520,158.414
C07166=1030.962,189.612,390.690,169.527,44.522,158.414
C07167=1030.957,189.363,390.714,169.523,44.523,158.414
C07168=1030.951,189.115,390.738,169.520,44.525,158.414
C07169=1030.944,188.831,390.765,169.516,44.527,158.414
C07170=1030.937,188.548,390.793,169.512,44.529,158.415
C07171=1030.931,188.264,390.820,169.509,44.531,158.415
C07172=1030.924,187.980,390.848,169.505,44.533,158.415
C07173=1030.918,187.732,390.872,169.501,44.535,158.415
C07174=1030.911,187.483,390.896,169.498,44.536,158.415
C07175=1030.906,187.234,390.919,169.495,44.538,158.415
C07176=1030.900,186.985,390.943,169.491,44.540,158.415
C07177=1030.894,186.736,390.967,169.489,44.542,158.415
C07178=1030.888,186.488,390.991,169.485,44.543,158.415
C07179=1030.882,186.238,391.016,169.482,44.545,158.415
C07180=1030.877,185.990,391.039,169.478,44.546,158.415
C07181=1030.870,185.741,391.062,169.475,44.549,158.415
C07182=1030.865,185.492,391.087,169.472,44.550,158.415
C07183=1030.859,185.244,391.111,169.468,44.552,158.415
C07184=1030.854,184.995,391.134,169.466,44.553,158.415
C07185=1030.847,184.746,391.158,169.462,44.555,158.415
C07186=1030.842,184.497,391.182,169.458,44.557,158.415
C07187=1030.836,184.249,391.206,169.456,44.559,158.415
C07188=1030.829,183.999,391.229,169.452,44.560,158.415
C07189=1030.824,183.751,391.254,169.449,44.562,158.415
C07190=1030.818,183.502,391.277,169.445,44.564,158.415
C07191=1030.813,183.253,391.301,169.442,44.566,158.415
C07192=1030.806,183.004,391.325,169.439,44.567,158.415
C07193=1030.800,182.756,391.349,169.435,44.569,158.415
C07194=1030.795,182.507,391.371,169.433,44.571,158.416
C07195=1030.788,182.257,391.395,169.429,44.573,158.416
C07196=1030.781,182.009,391.418,169.426,44.575,158.416
C07197=1030.776,181.760,391.441,169.423,44.577,158.416
C07198=1030.769,181.511,391.465,169.419,44.579,158.416
C07199=1030.763,181.263,391.488,169.416,44.581,158.416
C07200=1030.758,181.014,391.511,169.413,44.583,158.416
C07201=1030.751,180.765,391.535,169.410,44.585,158.416
C07202=1030.744,180.516,391.557,169.406,44.587,158.416
C07203=1030.739,180.267,391.580,169.403,44.588,158.416
C07204=1030.732,180.018,391.604,169.400,44.591,158.416
C07205=1030.726,179.769,391.627,169.396,44.593,158.417
C07206=1030.720,179.521,391.651,169.394,44.595,158.417
C07207=1030.714,179.271,391.674,169.390,44.597,158.417
C07208=1030.708,179.023,391.696,169.387,44.599,158.417
C07209=1030.702,178.774,391.719,169.384,44.601,158.417
C07210=1030.696,178.526,391.743,169.380,44.602,158.417
C07211=1030.689,178.276,391.766,169.377,44.604,158.417
C07212=1030.684,178.027,391.789,169.374,44.606,158.417
C07213=1030.677,177.779,391.812,169.370,44.608,158.417
C07214=1030.671,177.530,391.835,169.368,44.610,158.417
C07215=1030.665,177.281,391.859,169.364,44.613,158.417
C07216=1030.659,177.032,391.881,169.362,44.614,158.418
C07217=1030.653,176.783,391.904,169.358,44.616,158.418
C07218=1030.647,176.535,391.927,169.355,44.618,158.418
C07219=1030.640,176.285,391.951,169.352,44.620,158.418
C07220=1030.635,176.036,391.974,169.348,44.622,158.418
C07221=1030.629,175.788,391.997,169.346,44.624,158.418
C07222=1030.623,175.539,392.020,169.342,44.626,158.418
C07223=1030.616,175.291,392.043,169.339,44.628,158.418
C07224=1030.610,175.041,392.066,169.336,44.630,158.418
C07225=1030.604,174.792,392.089,169.333,44.632,158.418
C07226=1030.599,174.543,392.112,169.329,44.634,158.418
C07227=1030.593,174.294,392.135,169.326,44.636,158.419
C07228=1030.586,174.046,392.157,169.323,44.638,158.419
C07229=1030.581,173.797,392.180,169.320,44.640,158.419
C07230=1030.574,173.548,392.204,169.317,44.642,158.419
C07231=1030.568,173.299,392.227,169.314,44.644,158.419
C07232=1030.563,173.050,392.250,169.311,44.646,158.419
C07233=1030.556,172.766,392.276,169.307,44.648,158.419
C07234=1030.549,172.483,392.302,169.304,44.650,158.419
C07235=1030.542,172.199,392.328,169.300,44.652,158.419
C07236=1030.535,171.914,392.354,169.297,44.655,158.420
C07237=1030.529,171.665,392.377,169.293,44.657,158.420
C07238=1030.524,171.417,392.400,169.291,44.659,158.420
C07239=1030.517,171.168,392.422,169.287,44.661,158.420
C07240=1030.511,170.919,392.445,169.284,44.663,158.420
C07241=1030.506,170.670,392.468,169.281,44.665,158.420
C07242=1030.499,170.421,392.491,169.278,44.667,158.420
C07243=1030.494,170.172,392.514,169.275,44.669,158.420
C07244=1030.487,169.923,392.537,169.272,44.671,158.420
C07245=1030.481,169.674,392.560,169.269,44.673,158.421
C07246=1030.476,169.425,392.582,169.266,44.674,158.421
C07247=1030.470,169.176,392.605,169.262,44.676,158.421
C07248=1030.463,168.928,392.628,169.260,44.678,158.421
C07249=1030.458,168.679,392.651,169.256,44.681,158.421
C07250=1030.452,168.430,392.674,169.254,44.682,158.421
C07251=1030.446,168.181,392.697,169.250,44.685,158.421
C07252=1030.440,167.933,392.719,169.247,44.687,158.421
C07253=1030.434,167.683,392.741,169.244,44.689,158.421
C07254=1030.429,167.434,392.764,169.241,44.691,158.421
C07255=1030.423,167.185,392.787,169.239,44.693,158.422
C07256=1030.416,166.937,392.809,169.235,44.695,158.422
C07257=1030.411,166.688,392.832,169.233,44.697,158.422
C07258=1030.405,166.439,392.855,169.229,44.698,158.422
C07259=1030.399,166.190,392.878,169.226,44.700,158.422
C07260=1030.393,165.941,392.900,169.223,44.702,158.422
C07261=1030.387,165.692,392.923,169.220,44.704,158.422
C07262=1030.382,165.443,392.946,169.217,44.706,158.422
C07263=1030.376,165.194,392.969,169.214,44.708,158.422
C07264=1030.369,164.945,392.991,169.211,44.710,158.423
C07265=1030.364,164.696,393.013,169.208,44.712,158.423
C07266=1030.358,164.447,393.036,169.205,44.714,158.423
C07267=1030.353,164.199,393.059,169.202,44.716,158.423
C07268=1030.347,163.950,393.081,169.199,44.718,158.423
C07269=1030.341,163.701,393.104,169.197,44.720,158.423
C07270=1030.335,163.452,393.126,169.193,44.722,158.423
C07271=1030.330,163.203,393.149,169.190,44.724,158.423
C07272=1030.323,162.954,393.172,169.188,44.726,158.423
C07273=1030.318,162.705,393.194,169.184,44.728,158.423
C07274=1030.312,162.456,393.217,169.181,44.730,158.424
C07275=1030.306,162.207,393.239,169.178,44.732,158.424
C07276=1030.300,161.958,393.262,169.175,44.734,158.424
C07277=1030.295,161.710,393.284,169.173,44.736,158.424
